(* CODESYS project fablewhole.project
   CompiledLibraryCompatibilityVersion: LeadSysStudio V3.5 SP15 Patch 4
   Title: fablewhole

Project tree, tasks and I/O mapping:
  Device : MC508, Leadshine Technology Co., Ltd., order no. 508101, version 3.5.15.40
      settings: RetainMode = 0; RetainStartAddr = 20480; RetainEndAddr = 524287; RetainSize = 524288; LMMVersion = 0
    application Application
      libraries: Standard, * (System); Util, * (System)
      task T_Motion (cyclic, interval t#4ms, priority 1) calls PRG_Motion
      task T_App (cyclic, interval 20 ms, priority 8) calls PRG_IoMap, PRG_Supervisor, PRG_JobExec, PRG_Test, PRG_Carousels, PRG_Heating, PRG_Sim, PRG_Alarms
      task EtherCAT_Master_Leadshine_A (cyclic, interval 4000 µs, priority 0) calls EtherCAT_Master_Leadshine_A.EtherCAT_Task
      task T_Comms (cyclic, interval 100 ms, priority 15) calls PRG_GatewayComms, PRG_HMI, PRG_HACCP
      01_DUTs/
        data type E_MachMode
        data type E_Item
        data type E_GriddleState
        data type E_FaultClass
        data type ST_Recipe
        data type ST_PattyJob
        data type ST_GriddleSts
        data type ST_TrayInfo
        data type ST_GwCmd
        data type ST_GwAck
        data type ST_AxisSts
        data type ST_HeatZone
        data type ST_Alarm
        data type ST_HaccpRec
        data type ST_MechCmd
      00_GVLs/
        global variables GVL_Cfg
        global variables GVL_Par
        global variables GVL_IO
        global variables GVL_Axes
        global variables GVL_Cmd
        global variables GVL_Sts
        global variables GVL_Alm
        global variables GVL_Mech
      02_L1_Drivers/
        function F_Err [ST]
        function F_RaiseAlarm [ST]
        function block FB_AxisCtrl [ST]
        function block FB_PidHeater [ST]
        function block FB_PneuActuator [ST]
        function block FB_PressDrive [ST]
        function block FB_SensorIn [ST]
        function block FB_VfdIndex [ST]
      03_L2_Mechanisms/
        function block FB_Airlock [ST]
        function block FB_Fork [ST]
        function block FB_FridgeCarousel [ST]
        function block FB_Gantry [ST]
        function block FB_GriddleCarousel [ST]
        function block FB_Gripper [ST]
        function block FB_HeatBank [ST]
        function block FB_IKTransform [ST]
        function block FB_Press [ST]
        function block FB_Refrigeration [ST]
        function block FB_Scraper [ST]
      05_L4_Comms/
        program PRG_Alarms [ST]
        program PRG_GatewayComms [ST]
        program PRG_HACCP [ST]
        program PRG_HMI [ST]
      04_L3_Coordination/
        function block FB_GriddleTracker [ST]
        function block FB_HomingManager [ST]
        function block FB_JobQueue [ST]
        program PRG_JobExec [ST]
        program PRG_Supervisor [ST]
      06_Wiring_Sim_Test/
        program PRG_Carousels [ST]
        program PRG_Heating [ST]
        program PRG_IoMap [ST]
        program PRG_Motion [ST]
        program PRG_Sim [ST]
        program PRG_Test [ST]
    Device Diagnose
    Network Configuration
      LocalBus Config
    Resource Usage
    SoftMotion General Axis Pool
    High_Speed_IO_Module : High Speed IO, Leadshine Technology Co., Ltd., version 3.5.15.40
        unmapped channels: Genral_IO_IN, Genral_IO_Out
    LocalBus_Master_Module : LocalBus Master, Leadshine Technology Co., Ltd., version 3.5.15.40
    EtherCAT_Master_Leadshine_A : EtherCAT Master SoftMotion, 3S - Smart Software Solutions GmbH, version 3.5.15.30
        settings: NetworkName = 'ecat'; SelectNetworkByName = TRUE
      CS3E_D1008 : CS3E-D1008(COE), Leadshine Technology Co.,Ltd., order no. CS3E-D1008, version Revision=16#00000001
          settings: DC sync0 cycletime = 4000; DC sync1 cycletime = 4000
          unmapped channels: Control Word, Profile Target Position, Touch Probe Function, Last Error Code, Status Word, Modes of Operation display, Position Actual Value, Touch Probe Status, Touch Probe 1 Positive Value, Digital Inputs
        Axis : Axis, 3S - Smart Software Solutions GmbH, order no. 0, version 4.6.1.0
            settings: wDriveID = 0; Commisioning.smci.Distance = 100; Commisioning.smci.Velocity = 100; AdrOffset_8010 = 4; BitOffset_8010 = 0; BitLength_8010 = 16; Address_8010 = '%QW2'; Type_8010 = 'UINT'; AddressPointer_8010 = ADR(%QW2); AdrOffset_8020 = 8; BitOffset_8020 = 0; BitLength_8020 = 32; Address_8020 = '%QD2'; Type_8020 = 'DINT'; AddressPointer_8020 = ADR(%QD2); AdrOffset_8030 = 4294967295; BitOffset_8030 = 0; BitLength_8030 = 0; Address_8030 = ''; Type_8030 = ''; AddressPointer_8030 = 0; AdrOffset_8040 = 4294967295; BitOffset_8040 = 0; BitLength_8040 = 0; Address_8040 = ''; Type_8040 = ''; AddressPointer_8040 = 0; AdrOffset_8050 = 4294967295; BitOffset_8050 = 0; BitLength_8050 = 0; Address_8050 = ''; Type_8050 = ''; AddressPointer_8050 = 0; AdrOffset_8060 = 12; BitOffset_8060 = 0; BitLength_8060 = 16; Address_8060 = '%QW6'; Type_8060 = 'UINT'; AddressPointer_8060 = ADR(%QW6); AdrOffset_8070 = 4294967295;
              BitOffset_8070 = 0; BitLength_8070 = 0; Address_8070 = ''; Type_8070 = ''; AddressPointer_8070 = 0; AdrOffset_8080 = 4294967295; BitOffset_8080 = 0; BitLength_8080 = 0; Address_8080 = ''; Type_8080 = ''; AddressPointer_8080 = 0; AdrOffset_8090 = 4294967295; BitOffset_8090 = 0; BitLength_8090 = 0; Address_8090 = ''; Type_8090 = ''; AddressPointer_8090 = 0; AdrOffset_8510 = 6; BitOffset_8510 = 0; BitLength_8510 = 16; Address_8510 = '%IW3'; Type_8510 = 'UINT'; AddressPointer_8510 = ADR(%IW3); AdrOffset_8520 = 12; BitOffset_8520 = 0; BitLength_8520 = 32; Address_8520 = '%ID3'; Type_8520 = 'DINT'; AddressPointer_8520 = ADR(%ID3); AdrOffset_8530 = 4294967295; BitOffset_8530 = 0; BitLength_8530 = 0; Address_8530 = ''; Type_8530 = ''; AddressPointer_8530 = 0; AdrOffset_8540 = 4294967295; BitOffset_8540 = 0; BitLength_8540 = 0; Address_8540 = ''; Type_8540 = '';
              AddressPointer_8540 = 0; AdrOffset_8550 = 8; BitOffset_8550 = 0; BitLength_8550 = 8; Address_8550 = '%IB8'; Type_8550 = 'SINT'; AddressPointer_8550 = ADR(%IB8); AdrOffset_8560 = 24; BitOffset_8560 = 0; BitLength_8560 = 32; Address_8560 = '%ID6'; Type_8560 = 'UDINT'; AddressPointer_8560 = ADR(%ID6); AdrOffset_8570 = 16; BitOffset_8570 = 0; BitLength_8570 = 16; Address_8570 = '%IW8'; Type_8570 = 'UINT'; AddressPointer_8570 = ADR(%IW8); AdrOffset_8580 = 20; BitOffset_8580 = 0; BitLength_8580 = 32; Address_8580 = '%ID5'; Type_8580 = 'DINT'; AddressPointer_8580 = ADR(%ID5); AdrOffset_8590 = 4294967295; BitOffset_8590 = 0; BitLength_8590 = 0; Address_8590 = ''; Type_8590 = ''; AddressPointer_8590 = 0; AdrOffset_8600 = 4294967295; BitOffset_8600 = 0; BitLength_8600 = 0; Address_8600 = ''; Type_8600 = ''; AddressPointer_8600 = 0; AdrOffset_8600 = 4294967295; BitOffset_8600 = 0; BitLength_8600 = 0;
              Address_8610 = ''; Type_8610 = ''; AddressPointer_8610 = 0; AdrOffset_8620 = 4294967295; BitOffset_8620 = 0; BitLength_8620 = 0; Address_8620 = ''; Type_8620 = ''; AddressPointer_8620 = 0
      CS3E_D1008_1 : CS3E-D1008(COE), Leadshine Technology Co.,Ltd., order no. CS3E-D1008, version Revision=16#00000001
          settings: DC sync0 cycletime = 4000; DC sync1 cycletime = 4000
          unmapped channels: Control Word, Profile Target Position, Touch Probe Function, Last Error Code, Status Word, Modes of Operation display, Position Actual Value, Touch Probe Status, Touch Probe 1 Positive Value, Digital Inputs
        Axis_1 : Axis, 3S - Smart Software Solutions GmbH, order no. 0, version 4.6.1.0
            settings: AdrOffset_8010 = 16; BitOffset_8010 = 0; BitLength_8010 = 16; Address_8010 = '%QW8'; Type_8010 = 'UINT'; AddressPointer_8010 = ADR(%QW8); AdrOffset_8020 = 20; BitOffset_8020 = 0; BitLength_8020 = 32; Address_8020 = '%QD5'; Type_8020 = 'DINT'; AddressPointer_8020 = ADR(%QD5); AdrOffset_8030 = 4294967295; BitOffset_8030 = 0; BitLength_8030 = 0; Address_8030 = ''; Type_8030 = ''; AddressPointer_8030 = 0; AdrOffset_8040 = 4294967295; BitOffset_8040 = 0; BitLength_8040 = 0; Address_8040 = ''; Type_8040 = ''; AddressPointer_8040 = 0; AdrOffset_8050 = 4294967295; BitOffset_8050 = 0; BitLength_8050 = 0; Address_8050 = ''; Type_8050 = ''; AddressPointer_8050 = 0; AdrOffset_8060 = 24; BitOffset_8060 = 0; BitLength_8060 = 16; Address_8060 = '%QW12'; Type_8060 = 'UINT'; AddressPointer_8060 = ADR(%QW12); AdrOffset_8070 = 4294967295; BitOffset_8070 = 0; BitLength_8070 = 0; Address_8070 = '';
              Type_8070 = ''; AddressPointer_8070 = 0; AdrOffset_8080 = 4294967295; BitOffset_8080 = 0; BitLength_8080 = 0; Address_8080 = ''; Type_8080 = ''; AddressPointer_8080 = 0; AdrOffset_8090 = 4294967295; BitOffset_8090 = 0; BitLength_8090 = 0; Address_8090 = ''; Type_8090 = ''; AddressPointer_8090 = 0; AdrOffset_8510 = 30; BitOffset_8510 = 0; BitLength_8510 = 16; Address_8510 = '%IW15'; Type_8510 = 'UINT'; AddressPointer_8510 = ADR(%IW15); AdrOffset_8520 = 36; BitOffset_8520 = 0; BitLength_8520 = 32; Address_8520 = '%ID9'; Type_8520 = 'DINT'; AddressPointer_8520 = ADR(%ID9); AdrOffset_8530 = 4294967295; BitOffset_8530 = 0; BitLength_8530 = 0; Address_8530 = ''; Type_8530 = ''; AddressPointer_8530 = 0; AdrOffset_8540 = 4294967295; BitOffset_8540 = 0; BitLength_8540 = 0; Address_8540 = ''; Type_8540 = ''; AddressPointer_8540 = 0; AdrOffset_8550 = 32; BitOffset_8550 = 0;
              BitLength_8550 = 8; Address_8550 = '%IB32'; Type_8550 = 'SINT'; AddressPointer_8550 = ADR(%IB32); AdrOffset_8560 = 48; BitOffset_8560 = 0; BitLength_8560 = 32; Address_8560 = '%ID12'; Type_8560 = 'UDINT'; AddressPointer_8560 = ADR(%ID12); AdrOffset_8570 = 40; BitOffset_8570 = 0; BitLength_8570 = 16; Address_8570 = '%IW20'; Type_8570 = 'UINT'; AddressPointer_8570 = ADR(%IW20); AdrOffset_8580 = 44; BitOffset_8580 = 0; BitLength_8580 = 32; Address_8580 = '%ID11'; Type_8580 = 'DINT'; AddressPointer_8580 = ADR(%ID11); AdrOffset_8590 = 4294967295; BitOffset_8590 = 0; BitLength_8590 = 0; Address_8590 = ''; Type_8590 = ''; AddressPointer_8590 = 0; AdrOffset_8600 = 4294967295; BitOffset_8600 = 0; BitLength_8600 = 0; Address_8600 = ''; Type_8600 = ''; AddressPointer_8600 = 0; AdrOffset_8600 = 4294967295; BitOffset_8600 = 0; BitLength_8600 = 0; Address_8610 = ''; Type_8610 = ''; AddressPointer_8610 = 0;
              AdrOffset_8620 = 4294967295; BitOffset_8620 = 0; BitLength_8620 = 0; Address_8620 = ''; Type_8620 = ''; AddressPointer_8620 = 0
    ModbusCOM_Master_1 : ModbusCOM RS-485 Master, Leadshine Technology Co., Ltd., version 3.5.15.40
        settings: com.Parity = 2; com.Baudrate = 115200
      ModbusCOM_Slave : ModbusCOM Slave, Leadshine Technology Co., Ltd., version 3.5.15.40
          settings: ModBusRTU_ErrorCode = 0; channel 00.FuncCode = 16; channel 00.ControlMode = 1; channel 00.ResendCount = 3; channel 00.WriteRegOffSet = 25089; channel 00.WriteRegLeg = 2; channel 00.IOChannel = 0; channel 00.ChannelName = 'pr0'; channel 00.ChannelNote = ''; channel 01.FuncCode = 16; channel 01.ControlMode = 1; channel 01.ResendCount = 3; channel 01.WriteRegOffSet = 25097; channel 01.WriteRegLeg = 2; channel 01.ChannelName = 'pr1'; channel 01.ChannelNote = ''; channel 02.FuncCode = 16; channel 02.ControlMode = 1; channel 02.ResendCount = 3; channel 02.WriteRegOffSet = 25105; channel 02.WriteRegLeg = 2; channel 02.IOChannel = 2; channel 02.ChannelName = 'pr2'; channel 02.ChannelNote = ''; channel 03.FuncCode = 6; channel 03.ControlMode = 1; channel 03.ResendCount = 1; channel 03.WriteRegOffSet = 24578; channel 03.IOChannel = 3; channel 03.ChannelName = 'hometrig'; channel 03.ChannelNote = ''; channel 04.FuncCode = 3; channel 04.ResendCount = 1; channel 04.ReadRegOffSet = 4099; channel 04.IOChannel = 4; channel 04.ChannelName = 'homestatus'; channel 04.ChannelNote = ''; channel 05.FuncCode = 6; channel 05.ControlMode = 1; channel 05.ResendCount = 1;
            channel 05.WriteRegOffSet = 6145; channel 05.IOChannel = 5; channel 05.ChannelName = 'jog'; channel 05.ChannelNote = ''; Vendor.ChannelNum = 6; Vendor.Timeout = 200
          unmapped channels: ErrorCode, channel 00, channel 00, channel 00, channel 01, channel 01, channel 01, channel 02, channel 02, channel 02, channel 03, channel 03, channel 03, channel 04, channel 04, channel 05, channel 05, channel 05
      ModbusCOM_Slave_1 : ModbusCOM Slave, Leadshine Technology Co., Ltd., version 3.5.15.40
          settings: ModBusRTU_ErrorCode = 0; Vendor.SlaveID = 2
          unmapped channels: ErrorCode
      ModbusCOM_Slave_2 : ModbusCOM Slave, Leadshine Technology Co., Ltd., version 3.5.15.40
          settings: ModBusRTU_ErrorCode = 0; Vendor.SlaveID = 3
          unmapped channels: ErrorCode
      ModbusCOM_Slave_3 : ModbusCOM Slave, Leadshine Technology Co., Ltd., version 3.5.15.40
          settings: ModBusRTU_ErrorCode = 0; Vendor.SlaveID = 4
          unmapped channels: ErrorCode
    ModbusTCP_Slave_Device : Modbus TCP Slave, Leadshine Technology Co., Ltd., version 00.00.00.10
*)

// Device/Application/01_DUTs/E_MachMode
{attribute 'qualified_only'}
{attribute 'strict'}
TYPE E_MachMode :
(
    BOOT    := 0,
    HOMING  := 1,
    READY   := 2,
    RUN     := 3,
    CLEAN   := 4,
    FAULT   := 5,
    ESTOP   := 6
);
END_TYPE

// Device/Application/01_DUTs/E_Item
{attribute 'qualified_only'}
{attribute 'strict'}
TYPE E_Item :
(
    NONE      := 0,
    BEEF      := 1,
    CHICKEN   := 2,
    BACON     := 3,
    PINEAPPLE := 4
);
END_TYPE

// Device/Application/01_DUTs/E_GriddleState
{attribute 'qualified_only'}
{attribute 'strict'}
TYPE E_GriddleState :
(
    EMPTY           := 0,
    LOADING         := 1,
    COOKING         := 2,
    READY_TO_SCRAPE := 3,
    SCRAPING        := 4,
    FAULTED         := 5
);
END_TYPE

// Device/Application/01_DUTs/E_FaultClass
{attribute 'qualified_only'}
{attribute 'strict'}
TYPE E_FaultClass :
(
    INFO         := 0,
    QUARANTINE   := 1,
    ZONE_STOP    := 2,
    MACHINE_STOP := 3
);
END_TYPE

// Device/Application/01_DUTs/ST_Recipe
TYPE ST_Recipe :
STRUCT
    item        : UINT;           // E_Item value
    cookTimeS   : LREAL := 90.0;
    smashDurS   : LREAL := 8.0;
    smashPosMm  : LREAL := 4.0;   // platen gap at smash
    holdPosMm   : LREAL := 6.0;   // light-contact gap for remainder of cook
    platenSetC  : LREAL := 200.0;
END_STRUCT
END_TYPE

// Device/Application/01_DUTs/ST_PattyJob
TYPE ST_PattyJob :
STRUCT
    jobId     : UDINT;
    orderId   : UDINT;
    item      : UINT;
    trayId    : UINT;
    griddleId : INT;
    slot      : INT;
END_STRUCT
END_TYPE

// Device/Application/01_DUTs/ST_GriddleSts
TYPE ST_GriddleSts :
STRUCT
    state        : UINT;   // E_GriddleState value
    item         : UINT;
    count        : INT;
    cookElapsedS : LREAL;
    batchId      : UDINT;
END_STRUCT
END_TYPE

// Device/Application/01_DUTs/ST_TrayInfo
TYPE ST_TrayInfo :
STRUCT
    trayId    : UINT;
    item      : UINT;
    remaining : INT;
    level     : INT;   // 0..19
    face      : INT;   // 0..1
    inChamber : BOOL;
END_STRUCT
END_TYPE

// Device/Application/01_DUTs/ST_GwCmd
TYPE ST_GwCmd :
STRUCT
    seq  : UINT;
    code : UINT;    // see GVL_Cfg CMD_* constants
    p1   : DINT;
    p2   : DINT;
    p3   : DINT;
    p4   : DINT;
END_STRUCT
END_TYPE

// Device/Application/01_DUTs/ST_GwAck
TYPE ST_GwAck :
STRUCT
    seqEcho : UINT;
    busy    : BOOL;
    done    : BOOL;
    error   : BOOL;
    errorId : UDINT;
END_STRUCT
END_TYPE

// Device/Application/01_DUTs/ST_AxisSts
TYPE ST_AxisSts :
STRUCT
    powered : BOOL;
    homed   : BOOL;
    inPos   : BOOL;
    actPos  : LREAL;
    errorId : UDINT;
END_STRUCT
END_TYPE

// Device/Application/01_DUTs/ST_HeatZone
TYPE ST_HeatZone :
STRUCT
    setC    : LREAL;
    actC    : LREAL;
    outPct  : LREAL;
    tcOk    : BOOL;
    atSet   : BOOL;
    enabled : BOOL;
END_STRUCT
END_TYPE

// Device/Application/01_DUTs/ST_Alarm
TYPE ST_Alarm :
STRUCT
    id     : UDINT;      // (subsystem<<16) OR code
    class  : UINT;       // E_FaultClass value
    tsS    : UDINT;      // uptime seconds at raise
    active : BOOL;
    acked  : BOOL;
END_STRUCT
END_TYPE

// Device/Application/01_DUTs/ST_HaccpRec
TYPE ST_HaccpRec :
STRUCT
    batchId    : UDINT;
    item       : UINT;
    griddleId  : INT;
    platenTopC : LREAL;
    platenBotC : LREAL;
    cookS      : LREAL;
    tStartS    : UDINT;
    tEndS      : UDINT;
    result     : UINT;   // 0=OK 1=QUARANTINE
END_STRUCT
END_TYPE

// Device/Application/01_DUTs/ST_MechCmd
TYPE ST_MechCmd :
STRUCT
    code : UINT;    // mechanism-local, see GVL_Cfg MCMD_* constants
    p1   : LREAL;
    p2   : LREAL;
    p3   : LREAL;
END_STRUCT
END_TYPE

// Device/Application/00_GVLs/GVL_Cfg
(* ============================================================
   GVL_Cfg — machine constants. VAR_GLOBAL CONSTANT.
   SIM_MODE is the ONLY switch between simulation and hardware.
   Set FALSE for production download. Never change at runtime.
   ============================================================ *)
VAR_GLOBAL CONSTANT
    SIM_MODE          : BOOL  := TRUE;    // <<< FALSE for real hardware
    SIM_TIME_SCALE    : LREAL := 5.0;     // thermal/cook acceleration in sim (1.0 = real time)

    T_MOTION_MS       : LREAL := 4.0;
    T_APP_MS          : LREAL := 20.0;

    // ---- Counts & geometry ----
    GRIDDLE_COUNT       : INT := 4;
    PATTIES_PER_GRIDDLE : INT := 6;
    STATIONS            : INT := 4;       // carousel stations
    STATION_LOAD        : INT := 0;       // station index where loading happens
    STATION_SCRAPE      : INT := 2;       // opposite station
    TRAY_COLS           : INT := 6;
    TRAY_ROWS           : INT := 4;
    PATTIES_PER_TRAY    : INT := 24;
    TRAY_LEVELS         : INT := 20;
    TRAY_FACES          : INT := 2;

    // ---- Gantry kinematics (mm / deg) ----
    ARM_LEN     : LREAL := 350.0;
    GX_MIN      : LREAL := 0.0;
    GX_MAX      : LREAL := 900.0;
    THETA_MIN   : LREAL := -90.0;
    THETA_MAX   : LREAL := 90.0;
    GZ_UP       : LREAL := 0.0;
    GZ_PICK     : LREAL := 80.0;
    GZ_PLACE    : LREAL := 60.0;
    THETA_SAFE  : LREAL := 0.0;
    GX_PARK     : LREAL := 50.0;
    // tray pick grid (chamber tray held by fork)
    PICK_BASE_X    : LREAL := 700.0;
    PICK_BASE_Y    : LREAL := -150.0;
    PICK_SPACING_X : LREAL := 60.0;
    PICK_SPACING_Y : LREAL := 60.0;
    // griddle place grid (station 0, bottom platen)
    PLACE_BASE_X   : LREAL := 450.0;
    PLACE_BASE_Y   : LREAL := 0.0;
    PLACE_SPC_X    : LREAL := 70.0;
    PLACE_SPC_Y    : LREAL := 70.0;
    PLACE_COLS     : INT   := 3;      // 3 x 2 slots on a griddle

    // ---- Speeds ----
    G_VEL      : LREAL := 400.0;   G_ACC : LREAL := 1500.0;   // gantry X mm/s
    T_VEL      : LREAL := 120.0;   T_ACC : LREAL := 500.0;    // theta deg/s
    Z_VEL      : LREAL := 200.0;   Z_ACC : LREAL := 1000.0;
    S_VEL      : LREAL := 300.0;   S_ACC : LREAL := 1200.0;   // scraper
    F_VEL      : LREAL := 150.0;   F_ACC : LREAL := 400.0;    // fork
    JOG_VEL_MAX: LREAL := 50.0;

    // ---- Recipe edit bounds (PRG_HMI rejects writes outside these) ----
    REC_COOK_MIN   : LREAL := 10.0;   REC_COOK_MAX   : LREAL := 300.0;  // s
    REC_SMDUR_MIN  : LREAL := 0.0;    REC_SMDUR_MAX  : LREAL := 30.0;   // s
    REC_SMPOS_MIN  : LREAL := 2.0;    REC_SMPOS_MAX  : LREAL := 12.0;   // mm gap
    REC_HLPOS_MIN  : LREAL := 3.0;    REC_HLPOS_MAX  : LREAL := 15.0;   // mm gap
    REC_PLSET_MIN  : LREAL := 120.0;  REC_PLSET_MAX  : LREAL := 230.0;  // degC

    // ---- Press PR path parameters ----
    PRESS_OPEN_MM     : LREAL := 60.0;  // path 0 open position (clamshell gap)
    PRESS_TRIM_MAX_MM : LREAL := 2.0;   // per-press calibration trim clamp (+/-)

    // ---- CS2RS press Modbus RTU parameterization (RS485, NetworkConfig channels) ----
    PRESS_BENCH_DRIVE : INT := 0;      // bench: -1 = none; 0..3 = that press drive runs
                                        // REAL (DI motion + Modbus params) while machine is sim
    PRESS_PULSES_PER_MM : LREAL := 1000.0;  // TODO calibrate: drive gear -> pulses per mm gap
    // Channel setup reference (VERIFIED against CS2RS manual 5.4.1) — the
    // registers live in the NetworkConfig channel config, not in code:
    //   write-multiple (FC16), length 2, per path: 0x6201 (path0 pos H/L),
    //   0x6209 (path1), 0x6211 (path2). Trigger reg 0x6002 (unused; DI does motion).

    // ---- Scraper geometry ----
    SC_ENGAGE_Z   : LREAL := 45.0;
    SC_UP_Z       : LREAL := 0.0;
    SC_SWEEP_X0   : LREAL := 100.0;
    SC_SWEEP_X1   : LREAL := 420.0;
    SC_ROW_Y      : ARRAY[0..2] OF LREAL := [0.0, 70.0, 140.0];
    SC_STROKES    : INT := 3;

    // ---- Fork geometry ----
    FORK_LEVEL_H   : LREAL := 90.0;   // mm per tray level
    FORK_Z0        : LREAL := 50.0;
    FORK_MICROLIFT : LREAL := 8.0;
    FORK_TELE_OUT  : LREAL := 300.0;
    FORK_TELE_IN   : LREAL := 0.0;

    // ---- Carousels ----
    ENC_CPR          : DINT := 4096;          // counts per carousel rev
    IDX_SPEED_FAST   : INT  := 300;           // VFD speed ref (raw)
    IDX_SPEED_CREEP  : INT  := 40;
    IDX_DECEL_WIN    : DINT := 300;           // counts before target -> creep
    IDX_STOP_WIN     : DINT := 25;            // counts tolerance to drop pin
    IDX_VERIFY_WIN   : DINT := 40;            // encoder-vs-pin plausibility

    // ---- Heating ----
    HEAT_ZONES     : INT   := 8;
    PWM_WINDOW_MS  : LREAL := 2000.0;
    HEAT_KP        : LREAL := 4.0;
    HEAT_KI        : LREAL := 0.05;           // %/ (degC*s)
    HEAT_AT_BAND   : LREAL := 5.0;            // |err| <= band -> atSet
    HEAT_MAX_STAGGER : INT := 2;              // platens ramping at once
    TC_RATE_MAX    : LREAL := 8.0;            // degC/s plausibility
    FRIDGE_SET_C   : LREAL := 4.0;
    FRIDGE_HYST_C  : LREAL := 1.0;
    FRIDGE_EXC_S   : LREAL := 300.0;          // excursion > 5 min -> QUARANTINE

    // ---- Timeouts ----
    TO_AXIS_MOVE   : TIME := T#15S;
    TO_AXIS_HOME   : TIME := T#40S;
    TO_PNEU        : TIME := T#3S;
    TO_PRESS       : TIME := T#15S;
    TO_INDEX       : TIME := T#25S;
    TO_MECH        : TIME := T#60S;
    SCRAPE_GUARD_S : LREAL := 8.0;
    GW_TIMEOUT_S   : LREAL := 10.0;

    // ---- Command codes: Gateway -> PLC (ST_GwCmd.code) ----
    CMD_NOP         : UINT := 0;
    CMD_FETCH_TRAY  : UINT := 1;   // p1=item p2=level p3=face
    CMD_LOAD_GRIDDLE: UINT := 2;   // p1=griddleId p2=count p3=item
    CMD_SCRAPE      : UINT := 3;   // p1=griddleId
    CMD_RETURN_TRAY : UINT := 4;   // p1=level p2=face
    CMD_CLEAN_MODE  : UINT := 5;
    CMD_ABORT       : UINT := 6;

    // ---- Mechanism-local command codes (ST_MechCmd.code) ----
    MCMD_NONE     : UINT := 0;
    MCMD_HOME     : UINT := 1;
    MCMD_PARK     : UINT := 2;
    MCMD_PICK     : UINT := 10;  // gantry: p1=trayIdx(0..23)
    MCMD_PLACE    : UINT := 11;  // gantry: p1=slot(0..5)
    MCMD_SANITIZE : UINT := 13;
    MCMD_FETCH    : UINT := 20;  // fork: p1=level
    MCMD_RETURN   : UINT := 21;  // fork: p1=level
    MCMD_SWEEP    : UINT := 30;  // scraper: p1=strokeIdx(0..2)
    MCMD_PROFILE  : UINT := 40;  // press: recipe via SetRecipe inputs
    MCMD_OPEN     : UINT := 41;  // press open
    MCMD_GOTO     : UINT := 50;  // carousel: p1=station

    // ---- Subsystem IDs for ErrorID = SHL(ss,16) OR code ----
    SS_GANTRY_X  : UINT := 1;   SS_GANTRY_T : UINT := 2;   SS_GANTRY_Z : UINT := 3;
    SS_SCRAPER_X : UINT := 4;   SS_SCRAPER_Y: UINT := 5;   SS_SCRAPER_Z: UINT := 6;
    SS_FORK_Z    : UINT := 7;   SS_FORK_TELE: UINT := 8;
    SS_PRESS_0   : UINT := 10;  // press n -> 10+n
    SS_GRID_CAR  : UINT := 20;  SS_FRIDGE_CAR : UINT := 21;
    SS_HEAT_0    : UINT := 30;  // zone z -> 30+z
    SS_AIRLOCK   : UINT := 40;  SS_REFRIG   : UINT := 41;
    SS_GANTRY    : UINT := 45;  SS_SCRAPER  : UINT := 46;  SS_FORK : UINT := 47;
    SS_GRIPPER   : UINT := 48;
    SS_JOBEXEC   : UINT := 50;  SS_HOMING   : UINT := 51;
    SS_GWCOMMS   : UINT := 60;  SS_PNEU     : UINT := 61;  SS_SENSOR : UINT := 62;

    // ---- Generic error codes ----
    ERR_NONE      : UINT := 0;
    ERR_TIMEOUT   : UINT := 1;
    ERR_DRIVE     : UINT := 2;
    ERR_NOT_HOMED : UINT := 3;
    ERR_UNREACH   : UINT := 4;   // IK unreachable
    ERR_BAD_CMD   : UINT := 5;
    ERR_INTERLOCK : UINT := 6;
    ERR_PIN       : UINT := 7;   // pin/encoder mismatch
    ERR_SENSOR    : UINT := 8;
    ERR_TC        : UINT := 9;
    ERR_ABORTED   : UINT := 10;
    ERR_BUSY      : UINT := 11;
END_VAR

// Device/Application/00_GVLs/GVL_Par
(* ============================================================
   GVL_Par — retained tunables (recipes, offsets). HMI-writable
   through bounds-checked paths only (PRG_HMI / PRG_GatewayComms).
   ============================================================ *)
VAR_GLOBAL RETAIN
    // Index by E_Item value 0..4; [0] unused
    aRecipe : ARRAY[0..4] OF ST_Recipe :=
        [(item:=0),
         (item:=1, cookTimeS:=90.0,  smashDurS:=8.0, smashPosMm:=4.0, holdPosMm:=6.0, platenSetC:=200.0),  // BEEF
         (item:=2, cookTimeS:=110.0, smashDurS:=8.0, smashPosMm:=5.0, holdPosMm:=7.0, platenSetC:=200.0),  // CHICKEN (validate 74C core!)
         (item:=3, cookTimeS:=60.0,  smashDurS:=0.0, smashPosMm:=8.0, holdPosMm:=8.0, platenSetC:=190.0),  // BACON heat only
         (item:=4, cookTimeS:=45.0,  smashDurS:=0.0, smashPosMm:=8.0, holdPosMm:=8.0, platenSetC:=180.0)]; // PINEAPPLE
    jogVel        : LREAL := 20.0;
    pickOffsetX   : LREAL := 0.0;   // commissioning trims
    pickOffsetY   : LREAL := 0.0;
    placeOffsetX  : LREAL := 0.0;
    placeOffsetY  : LREAL := 0.0;
    // per-press smash/hold position trim, mm (+ = larger gap); HMI-adjustable,
    // clamped to +/- GVL_Cfg.PRESS_TRIM_MAX_MM in PRG_HMI
    pressTrimMm   : ARRAY[0..3] OF LREAL := [0.0, 0.0, 0.0, 0.0];
END_VAR

// Device/Application/00_GVLs/GVL_IO
(* ============================================================
   GVL_IO — the ONLY POU with physical addresses.
   SIM NOTE: in SIM_MODE these are never read/written (PRG_IoMap
   short-circuits). Addresses below are PLACEHOLDERS — replace
   with the real electrical map during panel design (see
   MIGRATION_GUIDE.md step 2) and keep wire numbers in comments.
   ============================================================ *)
VAR_GLOBAL
    // ---- Press drives 1..4 (CS2RS PR mode, DI wiring) ----
    qPressSel0    : ARRAY[0..3] OF BOOL;  // TODO real per-drive addresses
    qPressSel1    : ARRAY[0..3] OF BOOL;
    qPressCtrg    : ARRAY[0..3] OF BOOL;
    qPressEnable  : ARRAY[0..3] OF BOOL;
    iPressInPos   : ARRAY[0..3] OF BOOL;
    iPressAlarm   : ARRAY[0..3] OF BOOL;

    // ---- Pneumatics ----
    qDoorFridgeFront AT %QX4.0 : BOOL;
    qDoorFridgeSide  AT %QX4.1 : BOOL;
    qDoorChamber     AT %QX4.2 : BOOL;
    qPinGriddle      AT %QX4.3 : BOOL;
    qPinFridge       AT %QX4.4 : BOOL;
    qGripper         AT %QX4.5 : BOOL;
    iDoorFrFront_Op  AT %IX3.0 : BOOL;  iDoorFrFront_Cl AT %IX3.1 : BOOL;
    iDoorFrSide_Op   AT %IX3.2 : BOOL;  iDoorFrSide_Cl  AT %IX3.3 : BOOL;
    iDoorChamber_Op  AT %IX3.4 : BOOL;  iDoorChamber_Cl AT %IX3.5 : BOOL;
    iPinGriddle_Ext  AT %IX3.6 : BOOL;  iPinGriddle_Ret AT %IX3.7 : BOOL;
    iPinFridge_Ext   AT %IX4.0 : BOOL;  iPinFridge_Ret  AT %IX4.1 : BOOL;
    iGripAcquired    AT %IX4.2 : BOOL;

    // ---- Carousel VFDs (hardwired run/dir + analog/comms speed) ----
    qGridCarFwd AT %QX5.0 : BOOL;  qGridCarRev AT %QX5.1 : BOOL;
    qFrCarFwd   AT %QX5.2 : BOOL;  qFrCarRev   AT %QX5.3 : BOOL;
    wGridCarSpeed AT %QW10 : INT;  wFrCarSpeed  AT %QW11 : INT;
    diGridCarEnc  AT %ID12 : DINT; diFrCarEnc   AT %ID14 : DINT;
    iGridCarHome  AT %IX5.0 : BOOL; iFrCarHome  AT %IX5.1 : BOOL;

    // ---- Heating (R2 modules) ----
    qSsr         : ARRAY[0..7] OF BOOL;
    wPlatenTemp AT %IW20  : ARRAY[0..7] OF INT;   // 0.1 degC
    wFridgeTemp AT %IW28  : INT;                  // 0.1 degC

    // ---- BENCH press-drive terminals (old-rig wiring; PRESS_BENCH_DRIVE=0) ----
    qBenchPrAdd0    AT %QX1.5 : BOOL;  // drive SI = ADD0 (ex Z_DO_Down)
    qBenchPrAdd1    AT %QX1.7 : BOOL;  // drive SI = ADD1 (rewired)
    qBenchPrCtrg    AT %QX1.6 : BOOL;  // drive SI = CTRG (ex Z_Trig)
    qBenchPrDisable AT %QX1.3 : BOOL;  // drive enable line, INVERTED: TRUE = disable (ex Z_Disable)
    iBenchPrInPos   AT %IX1.0 : BOOL;  // SO1 INP (ex Z_InPos)
    iBenchPrAlarm   AT %IX1.1 : BOOL;  // SO3 ALM (ex Z_Alarm — check polarity!)

    // ---- RS485 Modbus master channel image (press PR position writes) ----
    // PLACEHOLDER addresses: after creating the 3 write channels in
    // NetworkConfig (RS485 -> Modbus Master), set these to the addresses the
    // master's I/O mapping actually assigns (old-project pattern: data words
    // %QW, trigger bit %QX, done bit %IX, error word %IW).
    qMbPr0Data AT %QW13 : ARRAY[0..1] OF WORD;  // CH0: slave1 FC16 25089/0x6201 len2 (path0 pos H,L)
    qMbPr1Data AT %QW16 : ARRAY[0..1] OF WORD;  // CH1: slave1 FC16 25097/0x6209 len2 (path1)
    qMbPr2Data AT %QW19 : ARRAY[0..1] OF WORD;  // CH2: slave1 FC16 25105/0x6211 len2 (path2)
    qMbPr0Trig AT %QX30.0 : BOOL;               // trigger control bits
    qMbPr1Trig AT %QX36.0 : BOOL;
    qMbPr2Trig AT %QX42.0 : BOOL;
    iMbPr0Done AT %IX54.0 : BOOL;               // processing complete states
    iMbPr1Done AT %IX54.1 : BOOL;
    iMbPr2Done AT %IX54.2 : BOOL;
    iMbPrErr   AT %IW26   : WORD;               // master ErrorCode (0 = ok)
    // homing + status channels
    qMbPrHomeData AT %QW22   : WORD;            // CH3: slave1 FC06 0x6002/24578 len1 (0x0020 = home)
    qMbPrHomeTrig AT %QX46.0 : BOOL;
    iMbPrHomeDone AT %IX54.3 : BOOL;
    iMbPrStatus   AT %IW28   : WORD;            // CH4: slave1 FC03 0x1003/4099 len1, CYCLE 100ms
    // jog channel (mapped)
    qMbPrJogData AT %QW24   : WORD;             // CH5: slave1 FC06 0x1801/6145 len1 (0x4001/0x4002)
    qMbPrJogTrig AT %QX50.0 : BOOL;
    iMbPrJogDone AT %IX58.1 : BOOL;
                                                // bits: 0x01 fault 0x02 enabled 0x04 running
                                                //       0x20 path done 0x40 homing done

    // ---- Fork brake ----
    qForkBrakeRelease AT %QX7.0 : BOOL;
    iForkBrakeOk      AT %IX6.0 : BOOL;
    iForkTrayPresent  AT %IX6.1 : BOOL;

    // ---- Safety controller status (monitor only) ----
    iSafetyOk        AT %IX7.0 : BOOL;
    iZonePwrMotion   AT %IX7.1 : BOOL;
    iZonePwrPress    AT %IX7.2 : BOOL;
END_VAR

// Device/Application/00_GVLs/GVL_Axes
(* ============================================================
   GVL_Axes — SoftMotion axis references.
   SIMULATION BUILD: the dummy declarations below let the project
   compile with SM3_Basic present but no drives; FB_AxisCtrl never
   calls MC_* while SIM_MODE=TRUE.
   PRODUCTION BUILD: DELETE these dummies and pass the device-tree
   axis objects (names created by the EtherCAT config) directly in
   PRG_Motion — see MIGRATION_GUIDE.md step 3.
   ============================================================ *)
VAR_GLOBAL
    axRefGantryX  : AXIS_REF_SM3;
    axRefGantryT  : AXIS_REF_SM3;
    axRefGantryZ  : AXIS_REF_SM3;
    axRefScraperX : AXIS_REF_SM3;
    axRefScraperY : AXIS_REF_SM3;
    axRefScraperZ : AXIS_REF_SM3;
    axRefForkZ    : AXIS_REF_SM3;
    axRefForkTele : AXIS_REF_SM3;
END_VAR

// Device/Application/00_GVLs/GVL_Cmd
(* ============================================================
   GVL_Cmd — commands INTO the PLC (Gateway + HMI + test).
   Modbus-TCP register images live here (%MW). The MC508 Modbus
   TCP slave exposes %MW to the Gateway.
   ============================================================ *)
VAR_GLOBAL
    // Gateway command image (Modbus 40001..) — packed by PRG_GatewayComms
    mbCmdRegs AT %MW0  : ARRAY[0..9]  OF WORD;   // seq,code,p1..p4 (DINT lo/hi)
    mbAckRegs AT %MW10 : ARRAY[0..5]  OF WORD;
    mbStsRegs AT %MW20 : ARRAY[0..79] OF WORD;
    mbParRegs AT %MW500: ARRAY[0..59] OF WORD;

    gwCmd     : ST_GwCmd;        // decoded, latched command
    gwAck     : ST_GwAck;
    gwHeartbeatIn : UINT;        // written by Gateway (reg in mbCmdRegs[9])
    gwAlive   : BOOL;
    gwPending : BOOL;            // new latched command awaiting JobExec

    // HMI request bits (edge-processed in PRG_HMI)
    hmiStart, hmiStop, hmiReset, hmiAck, hmiClean : BOOL;
    hmiMaintPin : UINT;          // maintenance password value
    hmiJogAxis  : INT;           // 0=none 1..8
    hmiJogPlus, hmiJogMinus : BOOL;

    // HMI recipe editor (bounds-checked in PRG_HMI; rejected in RUN)
    hmiRecItem  : UINT;          // 1..4 = E_Item to edit
    hmiRecField : UINT;          // 1=cookTimeS 2=smashDurS 3=smashPosMm 4=holdPosMm 5=platenSetC
    hmiRecValue : LREAL;         // requested value
    hmiRecWrite : BOOL;          // rising edge applies
    hmiRecAck   : BOOL;          // feedback: accepted
    hmiRecErr   : BOOL;          // feedback: rejected (bounds / mode / index)

    // HMI press calibration trim (maintenance PIN required)
    hmiTrimPress : UINT;         // 0..3
    hmiTrimDelta : LREAL;        // +/- mm added to that press's trim
    hmiTrimWrite : BOOL;         // rising edge applies
    hmiTrimAck, hmiTrimErr : BOOL;

    // HMI press service commands (PIN-gated; bench/commissioning + maintenance)
    hmiPressSel   : UINT;        // 0..3
    hmiPressCmd   : UINT;        // 1=HOME 2=OPEN 3=PROFILE(uses hmiRecItem's recipe)
    hmiPressWrite : BOOL;        // rising edge executes
    hmiPressAck, hmiPressErr : BOOL;

    // LT2100E Modbus-TCP register image (see HMI_LT2100E_GUIDE.md)
    // HMI writes 600..609, reads 620..669. Packed/unpacked in PRG_HMI.
    hmiRegsCmd AT %MW600 : ARRAY[0..9]  OF WORD;
    hmiRegsSts AT %MW620 : ARRAY[0..49] OF WORD;

    // Processed requests to Supervisor
    reqStart, reqStop, reqReset, reqClean, reqAckAll : BOOL;

    // Test authority: PRG_Test drives mechanisms instead of JobExec
    testMode  : BOOL := TRUE;    // default TRUE in sim; set FALSE for gateway runs
    testStart : BOOL;            // rising edge starts the automated suite
END_VAR

// Device/Application/00_GVLs/GVL_Sts
(* ============================================================
   GVL_Sts — status OUT of the PLC + Supervisor coordination
   flags. Written by L2/L3 only; L4 reads.
   ============================================================ *)
VAR_GLOBAL
    mode        : E_MachMode := E_MachMode.BOOT;
    uptimeS     : UDINT;
    heartbeat   : UINT;
    // Supervisor coordination (read by owner PRGs each cycle)
    safetyOk    : BOOL;          // effective (sim: TRUE)
    enMotion    : BOOL;          // mechanisms may move
    enProcess   : BOOL;          // heat + refrigeration on
    abortAll    : BOOL;          // broadcast abort
    resetPulse  : BOOL;          // 1-cycle axis reset on FAULT->HOMING
    cleanCoolOk : BOOL;          // all platens < 60 C in CLEAN
    // Aggregates
    allHomed    : BOOL;
    heatAtSet   : BOOL;
    fridgeAtSet : BOOL;
    fridgeActC  : LREAL;
    aGriddle    : ARRAY[0..3] OF ST_GriddleSts;
    aHeat       : ARRAY[0..7] OF ST_HeatZone;
    tray        : ST_TrayInfo;
    pattyOnGriddle : ARRAY[0..3, 0..5] OF BOOL;  // process bookkeeping (v1: no optics)
    carGridStation : INT;
    carFridgeFace  : INT;
    haccpCount  : UDINT;
    lastHaccp   : ST_HaccpRec;
    activeAlarms: INT;
    gwSilent    : BOOL;
END_VAR

// Device/Application/00_GVLs/GVL_Alm
(* ============================================================
   GVL_Alm — alarm table + history. Managed by PRG_Alarms and
   F_RaiseAlarm (any POU may raise).
   ============================================================ *)
VAR_GLOBAL
    aActive  : ARRAY[0..63] OF ST_Alarm;
    nActive  : INT;
    worstClass : UINT;                 // highest active E_FaultClass
    reqZoneStop : BOOL;                // aggregated flags for Supervisor
    reqMachStop : BOOL;
END_VAR
VAR_GLOBAL RETAIN
    aHistory : ARRAY[0..199] OF ST_Alarm;
    histHead : INT;
END_VAR

// Device/Application/00_GVLs/GVL_Mech
(* ============================================================
   GVL_Mech — ALL FB instances live here (single ownership table).
   BODY-CALL OWNERSHIP (call the FB body ONLY in the listed PRG):
     PRG_Motion   (T_Motion): axis FBs, fbGantry, fbScraper, fbFork, fbGripper
     PRG_Carousels(T_App)   : press drives, presses, VFDs, carousels,
                              pneumatics, airlock
     PRG_Heating  (T_App)   : heaters, heat bank, refrigeration
   All other POUs only WRITE inputs / READ outputs of these instances.
   ============================================================ *)
VAR_GLOBAL
    // L1 axis drivers
    axGX, axGT, axGZ : FB_AxisCtrl;      // gantry X / theta / Z
    axSX, axSY, axSZ : FB_AxisCtrl;      // scraper
    axFZ, axFT       : FB_AxisCtrl;      // fork Z / telescope

    // L1 press drives + L2 presses
    drvPress : ARRAY[0..3] OF FB_PressDrive;
    fbPress  : ARRAY[0..3] OF FB_Press;

    // Pneumatics
    fbDoorFridgeFront, fbDoorFridgeSide, fbDoorChamber : FB_PneuActuator;
    fbPinGriddle, fbPinFridge, fbPneuGrip : FB_PneuActuator;

    // Carousels
    vfdGriddle, vfdFridge : FB_VfdIndex;
    fbGridCar  : FB_GriddleCarousel;
    fbFridgeCar: FB_FridgeCarousel;

    // Heating / cold
    fbHeater  : ARRAY[0..7] OF FB_PidHeater;
    fbHeatBank: FB_HeatBank;
    fbRefrig  : FB_Refrigeration;

    // Motion mechanisms
    fbIK      : FB_IKTransform;
    fbGripper : FB_Gripper;
    fbGantry  : FB_Gantry;
    fbScraper : FB_Scraper;
    fbFork    : FB_Fork;

    // Coordination
    fbAirlock : FB_Airlock;
    fbHoming  : FB_HomingManager;
    fbTracker : FB_GriddleTracker;
    fbQueue   : FB_JobQueue;
END_VAR

// Device/Application/06_Wiring_Sim_Test/PRG_Motion
(* ============================================================
   PRG_Motion — T_Motion (4 ms). Body-call owner for all axis FBs
   and the motion mechanisms. THE ONLY TASK TOUCHING MC_* / AXIS_REF.
   This is the ST equivalent of the CFC wiring diagram: pure
   parameter assignment + instance calls, no logic.
   MIGRATION: replace GVL_Axes.axRef* with the device-tree axis
   objects created by the EtherCAT scan (step 3 of the guide).
   ============================================================ *)
PROGRAM PRG_Motion
VAR
    init : BOOL;
END_VAR

IF NOT init THEN
    init := TRUE;
    GVL_Mech.axGX.SubsysId := GVL_Cfg.SS_GANTRY_X;   GVL_Mech.axGX.CycleMs := GVL_Cfg.T_MOTION_MS;
    GVL_Mech.axGT.SubsysId := GVL_Cfg.SS_GANTRY_T;   GVL_Mech.axGT.CycleMs := GVL_Cfg.T_MOTION_MS;
    GVL_Mech.axGZ.SubsysId := GVL_Cfg.SS_GANTRY_Z;   GVL_Mech.axGZ.CycleMs := GVL_Cfg.T_MOTION_MS;
    GVL_Mech.axSX.SubsysId := GVL_Cfg.SS_SCRAPER_X;  GVL_Mech.axSX.CycleMs := GVL_Cfg.T_MOTION_MS;
    GVL_Mech.axSY.SubsysId := GVL_Cfg.SS_SCRAPER_Y;  GVL_Mech.axSY.CycleMs := GVL_Cfg.T_MOTION_MS;
    GVL_Mech.axSZ.SubsysId := GVL_Cfg.SS_SCRAPER_Z;  GVL_Mech.axSZ.CycleMs := GVL_Cfg.T_MOTION_MS;
    GVL_Mech.axFZ.SubsysId := GVL_Cfg.SS_FORK_Z;     GVL_Mech.axFZ.CycleMs := GVL_Cfg.T_MOTION_MS;
    GVL_Mech.axFT.SubsysId := GVL_Cfg.SS_FORK_TELE;  GVL_Mech.axFT.CycleMs := GVL_Cfg.T_MOTION_MS;
END_IF

// ---- distribute enables / abort / reset ----
GVL_Mech.axGX.Sim := GVL_Cfg.SIM_MODE;  GVL_Mech.axGX.Enable := GVL_Sts.enMotion;
GVL_Mech.axGT.Sim := GVL_Cfg.SIM_MODE;  GVL_Mech.axGT.Enable := GVL_Sts.enMotion;
GVL_Mech.axGZ.Sim := GVL_Cfg.SIM_MODE;  GVL_Mech.axGZ.Enable := GVL_Sts.enMotion;
GVL_Mech.axSX.Sim := GVL_Cfg.SIM_MODE;  GVL_Mech.axSX.Enable := GVL_Sts.enMotion;
GVL_Mech.axSY.Sim := GVL_Cfg.SIM_MODE;  GVL_Mech.axSY.Enable := GVL_Sts.enMotion;
GVL_Mech.axSZ.Sim := GVL_Cfg.SIM_MODE;  GVL_Mech.axSZ.Enable := GVL_Sts.enMotion;
GVL_Mech.axFZ.Sim := GVL_Cfg.SIM_MODE;  GVL_Mech.axFZ.Enable := GVL_Sts.enMotion;
GVL_Mech.axFT.Sim := GVL_Cfg.SIM_MODE;  GVL_Mech.axFT.Enable := GVL_Sts.enMotion;
GVL_Mech.axGX.Abort := GVL_Sts.abortAll;  GVL_Mech.axGX.ResetExec := GVL_Sts.resetPulse;
GVL_Mech.axGT.Abort := GVL_Sts.abortAll;  GVL_Mech.axGT.ResetExec := GVL_Sts.resetPulse;
GVL_Mech.axGZ.Abort := GVL_Sts.abortAll;  GVL_Mech.axGZ.ResetExec := GVL_Sts.resetPulse;
GVL_Mech.axSX.Abort := GVL_Sts.abortAll;  GVL_Mech.axSX.ResetExec := GVL_Sts.resetPulse;
GVL_Mech.axSY.Abort := GVL_Sts.abortAll;  GVL_Mech.axSY.ResetExec := GVL_Sts.resetPulse;
GVL_Mech.axSZ.Abort := GVL_Sts.abortAll;  GVL_Mech.axSZ.ResetExec := GVL_Sts.resetPulse;
GVL_Mech.axFZ.Abort := GVL_Sts.abortAll;  GVL_Mech.axFZ.ResetExec := GVL_Sts.resetPulse;
GVL_Mech.axFT.Abort := GVL_Sts.abortAll;  GVL_Mech.axFT.ResetExec := GVL_Sts.resetPulse;

// ---- mechanism bodies (write axis inputs) ----
GVL_Mech.fbGripper(
    Sim  := GVL_Cfg.SIM_MODE,
    iAcquired := GVL_IO.iGripAcquired,
    Pneu := GVL_Mech.fbPneuGrip);

GVL_Mech.fbGantry(
    Enable := GVL_Sts.enMotion,
    Abort  := GVL_Sts.abortAll,
    Sim    := GVL_Cfg.SIM_MODE,
    AxX := GVL_Mech.axGX, AxT := GVL_Mech.axGT, AxZ := GVL_Mech.axGZ,
    Grip := GVL_Mech.fbGripper, IK := GVL_Mech.fbIK);

GVL_Mech.fbScraper(
    Enable := GVL_Sts.enMotion,
    Abort  := GVL_Sts.abortAll,
    Sim    := GVL_Cfg.SIM_MODE,
    AxX := GVL_Mech.axSX, AxY := GVL_Mech.axSY, AxZ := GVL_Mech.axSZ);

GVL_Mech.fbFork(
    Enable := GVL_Sts.enMotion,
    Abort  := GVL_Sts.abortAll,
    Sim    := GVL_Cfg.SIM_MODE,
    iBrakeOk := GVL_IO.iForkBrakeOk,
    iTrayPresent := GVL_IO.iForkTrayPresent,
    AxZ := GVL_Mech.axFZ, AxT := GVL_Mech.axFT);
IF NOT GVL_Cfg.SIM_MODE THEN
    GVL_IO.qForkBrakeRelease := GVL_Mech.fbFork.qBrakeRelease;
END_IF

// ---- axis bodies LAST (consume inputs written above) ----
GVL_Mech.axGX(Axis := GVL_Axes.axRefGantryX);
GVL_Mech.axGT(Axis := GVL_Axes.axRefGantryT);
GVL_Mech.axGZ(Axis := GVL_Axes.axRefGantryZ);
GVL_Mech.axSX(Axis := GVL_Axes.axRefScraperX);
GVL_Mech.axSY(Axis := GVL_Axes.axRefScraperY);
GVL_Mech.axSZ(Axis := GVL_Axes.axRefScraperZ);
GVL_Mech.axFZ(Axis := GVL_Axes.axRefForkZ);
GVL_Mech.axFT(Axis := GVL_Axes.axRefForkTele);

END_PROGRAM

// Device/Application/06_Wiring_Sim_Test/PRG_IoMap
(* ============================================================
   PRG_IoMap — T_App, runs FIRST. Housekeeping + the place for
   commissioning force-rungs (these networks become LD at the
   language refactor). All %I/%Q symbol reads/writes elsewhere go
   through the owner wiring PRGs; addresses exist ONLY in GVL_IO.
   ============================================================ *)
PROGRAM PRG_IoMap
VAR
    msAcc : LREAL;
END_VAR

msAcc := msAcc + GVL_Cfg.T_APP_MS;
IF msAcc >= 1000.0 THEN
    msAcc := msAcc - 1000.0;
    GVL_Sts.uptimeS := GVL_Sts.uptimeS + 1;
END_IF
// ---- bench press-drive terminal mapping (active when PRESS_BENCH_DRIVE = 0) ----
// Copies the unaddressed press-0 signal arrays to/from the physically wired
// bench terminals (declared in GVL_IO, old-rig addresses).
IF GVL_Cfg.PRESS_BENCH_DRIVE = 0 THEN
    GVL_IO.qBenchPrAdd0    := GVL_IO.qPressSel0[0];
    GVL_IO.qBenchPrAdd1    := GVL_IO.qPressSel1[0];
    GVL_IO.qBenchPrCtrg    := GVL_IO.qPressCtrg[0];
    GVL_IO.qBenchPrDisable := NOT GVL_IO.qPressEnable[0];   // wire is a DISABLE line
    GVL_IO.iPressInPos[0]  := GVL_IO.iBenchPrInPos;
    GVL_IO.iPressAlarm[0]  := GVL_IO.iBenchPrAlarm;         // if ALM is NC: invert here
END_IF

// TODO(commissioning): add per-signal force flags here, e.g.
//   IF forceDoorChamber THEN GVL_IO.qDoorChamber := forceVal; END_IF

END_PROGRAM

// Device/Application/04_L3_Coordination/PRG_Supervisor
(* ============================================================
   PRG_Supervisor — machine mode state machine (T_App, runs FIRST
   among coordinators). Owns: mode transitions, enable distribution,
   abort broadcast, homing orchestration, clean-mode thermal gate.
   Safety is only MONITORED here (GVL_Sts.safetyOk).
   ============================================================ *)
PROGRAM PRG_Supervisor
VAR
    rtStart, rtStop, rtReset, rtClean : R_TRIG;
    z          : INT;
    coolOk     : BOOL;
    firstScan  : BOOL := TRUE;
END_VAR

// effective safety status
GVL_Sts.safetyOk := GVL_Cfg.SIM_MODE OR GVL_IO.iSafetyOk;

rtStart(CLK := GVL_Cmd.reqStart);
rtStop (CLK := GVL_Cmd.reqStop);
rtReset(CLK := GVL_Cmd.reqReset);
rtClean(CLK := GVL_Cmd.reqClean);

// defaults each scan
GVL_Sts.resetPulse := FALSE;

// global overrides
IF NOT GVL_Sts.safetyOk THEN
    GVL_Sts.mode := E_MachMode.ESTOP;
END_IF
IF GVL_Alm.reqMachStop AND (GVL_Sts.mode <> E_MachMode.ESTOP) THEN
    GVL_Sts.mode := E_MachMode.FAULT;
END_IF

CASE GVL_Sts.mode OF
    E_MachMode.BOOT:
        GVL_Sts.enMotion := FALSE; GVL_Sts.enProcess := FALSE;
        GVL_Sts.abortAll := FALSE;
        IF GVL_Sts.safetyOk AND NOT firstScan THEN
            GVL_Sts.resetPulse := TRUE;
            GVL_Mech.fbHoming.Exec := TRUE;
            GVL_Sts.mode := E_MachMode.HOMING;
        END_IF

    E_MachMode.HOMING:
        GVL_Sts.enMotion := TRUE; GVL_Sts.enProcess := FALSE;
        IF GVL_Mech.fbHoming.Done THEN
            GVL_Mech.fbHoming.Exec := FALSE;
            GVL_Sts.mode := E_MachMode.READY;
        ELSIF GVL_Mech.fbHoming.Error THEN
            GVL_Mech.fbHoming.Exec := FALSE;
            GVL_Sts.mode := E_MachMode.FAULT;
        END_IF

    E_MachMode.READY:
        GVL_Sts.enMotion := TRUE; GVL_Sts.enProcess := TRUE;   // heat-up + pulldown
        IF GVL_Alm.reqZoneStop THEN
            GVL_Sts.mode := E_MachMode.FAULT;
        ELSIF rtStart.Q AND GVL_Sts.heatAtSet AND GVL_Sts.fridgeAtSet AND GVL_Sts.allHomed THEN
            GVL_Sts.mode := E_MachMode.RUN;
        END_IF

    E_MachMode.RUN:
        GVL_Sts.enMotion := TRUE; GVL_Sts.enProcess := TRUE;
        IF GVL_Alm.reqZoneStop THEN
            GVL_Sts.mode := E_MachMode.FAULT;
        ELSIF rtStop.Q THEN
            GVL_Sts.mode := E_MachMode.READY;      // finish-in-place is JobExec's job
        ELSIF rtClean.Q AND (GVL_Mech.fbQueue.Empty) THEN
            GVL_Sts.mode := E_MachMode.CLEAN;
        END_IF

    E_MachMode.CLEAN:
        GVL_Sts.enMotion := FALSE;                  // motion locked for operator
        GVL_Sts.enProcess := FALSE;                 // heaters off -> cool down
        coolOk := TRUE;
        FOR z := 0 TO 7 DO
            IF GVL_Sts.aHeat[z].actC >= 60.0 THEN coolOk := FALSE; END_IF
        END_FOR
        GVL_Sts.cleanCoolOk := coolOk;
        IF rtStart.Q AND coolOk THEN                // operator confirms clean done
            GVL_Sts.resetPulse := TRUE;
            GVL_Mech.fbHoming.Exec := TRUE;
            GVL_Sts.mode := E_MachMode.HOMING;
        END_IF

    E_MachMode.FAULT:
        GVL_Sts.enMotion := FALSE; GVL_Sts.enProcess := FALSE;
        GVL_Sts.abortAll := TRUE;
        IF rtReset.Q AND (NOT GVL_Alm.reqMachStop) AND (NOT GVL_Alm.reqZoneStop) THEN
            GVL_Sts.abortAll := FALSE;
            GVL_Sts.resetPulse := TRUE;
            GVL_Mech.fbHoming.Exec := TRUE;
            GVL_Sts.mode := E_MachMode.HOMING;
        END_IF

    E_MachMode.ESTOP:
        GVL_Sts.enMotion := FALSE; GVL_Sts.enProcess := FALSE;
        GVL_Sts.abortAll := TRUE;
        IF GVL_Sts.safetyOk AND rtReset.Q THEN
            GVL_Sts.abortAll := FALSE;
            GVL_Sts.resetPulse := TRUE;
            GVL_Mech.fbHoming.Exec := TRUE;
            GVL_Sts.mode := E_MachMode.HOMING;
        END_IF
END_CASE
firstScan := FALSE;

// homing manager body (same task, before PRG_Carousels)
GVL_Mech.fbHoming(
    Abort     := GVL_Sts.abortAll,
    Presses   := GVL_Mech.fbPress,
    Gantry    := GVL_Mech.fbGantry,
    Scraper   := GVL_Mech.fbScraper,
    Fork      := GVL_Mech.fbFork,
    GridCar   := GVL_Mech.fbGridCar,
    FridgeCar := GVL_Mech.fbFridgeCar);

// aggregates
GVL_Sts.allHomed := GVL_Mech.fbGantry.Homed AND GVL_Mech.fbScraper.Homed
                AND GVL_Mech.fbFork.Homed AND GVL_Mech.fbGridCar.Homed
                AND GVL_Mech.fbFridgeCar.Homed;
GVL_Sts.heatAtSet   := GVL_Mech.fbHeatBank.AllAtSet;
GVL_Sts.fridgeAtSet := GVL_Mech.fbRefrig.AtSet;
GVL_Sts.fridgeActC  := GVL_Mech.fbRefrig.ActC;

END_PROGRAM

// Device/Application/06_Wiring_Sim_Test/PRG_Carousels
(* ============================================================
   PRG_Carousels — T_App body-call owner: press drives, presses,
   pneumatics, VFD indexers, carousels, airlock. Pure wiring
   (the ST equivalent of a CFC sheet). Runs AFTER Supervisor/
   JobExec/Test (which write the Cmd inputs).
   ============================================================ *)
PROGRAM PRG_Carousels
VAR
    i    : INT;
    init : BOOL;
END_VAR

IF NOT init THEN
    init := TRUE;
    FOR i := 0 TO 3 DO
        GVL_Mech.drvPress[i].SubsysId := GVL_Cfg.SS_PRESS_0 + TO_UINT(i);
        GVL_Mech.fbPress[i].PressId := i;
    END_FOR
    GVL_Mech.fbDoorFridgeFront.SubsysId := GVL_Cfg.SS_AIRLOCK;
    GVL_Mech.fbDoorFridgeSide.SubsysId  := GVL_Cfg.SS_AIRLOCK;
    GVL_Mech.fbDoorChamber.SubsysId     := GVL_Cfg.SS_AIRLOCK;
    GVL_Mech.fbPinGriddle.SubsysId := GVL_Cfg.SS_GRID_CAR;
    GVL_Mech.fbPinFridge.SubsysId  := GVL_Cfg.SS_FRIDGE_CAR;
    GVL_Mech.fbPneuGrip.SubsysId   := GVL_Cfg.SS_GRIPPER;
    GVL_Mech.vfdGriddle.SubsysId := GVL_Cfg.SS_GRID_CAR;
    GVL_Mech.vfdFridge.SubsysId  := GVL_Cfg.SS_FRIDGE_CAR;
END_IF

// ---- presses ----
FOR i := 0 TO 3 DO
    GVL_Mech.fbPress[i].Enable := GVL_Sts.enMotion;
    GVL_Mech.fbPress[i].Abort  := GVL_Sts.abortAll;
    GVL_Mech.fbPress[i].Sim    := GVL_Cfg.SIM_MODE;
    GVL_Mech.fbPress[i].CycleMs:= GVL_Cfg.T_APP_MS;
    // bench override: the selected drive runs REAL while the machine is sim
    GVL_Mech.drvPress[i].Sim    := GVL_Cfg.SIM_MODE AND (i <> GVL_Cfg.PRESS_BENCH_DRIVE);
    GVL_Mech.drvPress[i].Enable := GVL_Sts.enMotion;
    GVL_Mech.drvPress[i].Abort  := GVL_Sts.abortAll;
    GVL_Mech.drvPress[i].CycleMs:= GVL_Cfg.T_APP_MS;
    GVL_Mech.drvPress[i].iInPos := GVL_IO.iPressInPos[i];
    GVL_Mech.drvPress[i].iAlarm := GVL_IO.iPressAlarm[i];
    GVL_Mech.fbPress[i](Drv := GVL_Mech.drvPress[i]);
    GVL_Mech.drvPress[i]();
    IF (NOT GVL_Cfg.SIM_MODE) OR (i = GVL_Cfg.PRESS_BENCH_DRIVE) THEN
        GVL_IO.qPressSel0[i]   := GVL_Mech.drvPress[i].qSel0;
        GVL_IO.qPressSel1[i]   := GVL_Mech.drvPress[i].qSel1;
        GVL_IO.qPressCtrg[i]   := GVL_Mech.drvPress[i].qCtrg;
        GVL_IO.qPressEnable[i] := GVL_Mech.drvPress[i].qEnable;
    END_IF
END_FOR

// ---- CS2RS Modbus PR-write transport: NetworkConfig channel routing ----
// Channels are created in NetworkConfig (RS485 -> Modbus Master), one
// write-multiple channel per PR path (see GVL_IO placeholders + GVL_Cfg
// reference). This glue routes the bench/press-0 drive's path-write request
// to the matching channel. Extend with channel banks for drives 1..3 when
// the full RS485 bus exists.
IF (NOT GVL_Cfg.SIM_MODE) OR (GVL_Cfg.PRESS_BENCH_DRIVE >= 0) THEN
    GVL_IO.qMbPr0Trig := FALSE;
    GVL_IO.qMbPr1Trig := FALSE;
    GVL_IO.qMbPr2Trig := FALSE;
    GVL_Mech.drvPress[0].MbWrDone := FALSE;
    GVL_Mech.drvPress[0].MbWrErr  := FALSE;
    CASE GVL_Mech.drvPress[0].MbPath OF
        0:  GVL_IO.qMbPr0Data[0] := GVL_Mech.drvPress[0].MbValH;
            GVL_IO.qMbPr0Data[1] := GVL_Mech.drvPress[0].MbValL;
            GVL_IO.qMbPr0Trig    := GVL_Mech.drvPress[0].MbWrExec;
            GVL_Mech.drvPress[0].MbWrDone := GVL_IO.iMbPr0Done AND GVL_Mech.drvPress[0].MbWrExec;
        1:  GVL_IO.qMbPr1Data[0] := GVL_Mech.drvPress[0].MbValH;
            GVL_IO.qMbPr1Data[1] := GVL_Mech.drvPress[0].MbValL;
            GVL_IO.qMbPr1Trig    := GVL_Mech.drvPress[0].MbWrExec;
            GVL_Mech.drvPress[0].MbWrDone := GVL_IO.iMbPr1Done AND GVL_Mech.drvPress[0].MbWrExec;
        2:  GVL_IO.qMbPr2Data[0] := GVL_Mech.drvPress[0].MbValH;
            GVL_IO.qMbPr2Data[1] := GVL_Mech.drvPress[0].MbValL;
            GVL_IO.qMbPr2Trig    := GVL_Mech.drvPress[0].MbWrExec;
            GVL_Mech.drvPress[0].MbWrDone := GVL_IO.iMbPr2Done AND GVL_Mech.drvPress[0].MbWrExec;
    END_CASE
    GVL_Mech.drvPress[0].MbWrErr :=
        (GVL_IO.iMbPrErr <> 0) AND GVL_Mech.drvPress[0].MbWrExec;
    // homing channel (FC06: 0x0020 -> 0x6002) + cyclic status word (0x1003)
    GVL_IO.qMbPrHomeData := 16#0020;
    GVL_IO.qMbPrHomeTrig := GVL_Mech.drvPress[0].MbHomeExec;
    GVL_Mech.drvPress[0].MbHomeDone :=
        GVL_IO.iMbPrHomeDone AND GVL_Mech.drvPress[0].MbHomeExec;
    GVL_Mech.drvPress[0].iStatusWord := GVL_IO.iMbPrStatus;
    // jog channel (FC06: 0x4001/0x4002 -> 0x1801)
    GVL_IO.qMbPrJogData := GVL_Mech.drvPress[0].MbJogVal;
    GVL_IO.qMbPrJogTrig := GVL_Mech.drvPress[0].MbJogExec;
    GVL_Mech.drvPress[0].MbJogDone :=
        GVL_IO.iMbPrJogDone AND GVL_Mech.drvPress[0].MbJogExec;
END_IF

// ---- pneumatics ----
GVL_Mech.fbDoorFridgeSide(Sim := GVL_Cfg.SIM_MODE, CycleMs := GVL_Cfg.T_APP_MS,
    iExtended := GVL_IO.iDoorFrSide_Op, iRetracted := GVL_IO.iDoorFrSide_Cl);
GVL_Mech.fbDoorChamber(Sim := GVL_Cfg.SIM_MODE, CycleMs := GVL_Cfg.T_APP_MS,
    iExtended := GVL_IO.iDoorChamber_Op, iRetracted := GVL_IO.iDoorChamber_Cl);
GVL_Mech.fbDoorFridgeFront(Sim := GVL_Cfg.SIM_MODE, CycleMs := GVL_Cfg.T_APP_MS,
    iExtended := GVL_IO.iDoorFrFront_Op, iRetracted := GVL_IO.iDoorFrFront_Cl);
GVL_Mech.fbPinGriddle(Sim := GVL_Cfg.SIM_MODE, CycleMs := GVL_Cfg.T_APP_MS,
    iExtended := GVL_IO.iPinGriddle_Ext, iRetracted := GVL_IO.iPinGriddle_Ret);
GVL_Mech.fbPinFridge(Sim := GVL_Cfg.SIM_MODE, CycleMs := GVL_Cfg.T_APP_MS,
    iExtended := GVL_IO.iPinFridge_Ext, iRetracted := GVL_IO.iPinFridge_Ret);
GVL_Mech.fbPneuGrip(Sim := GVL_Cfg.SIM_MODE, CycleMs := GVL_Cfg.T_APP_MS,
    iExtended := GVL_IO.iGripAcquired, iRetracted := NOT GVL_IO.iGripAcquired);
IF NOT GVL_Cfg.SIM_MODE THEN
    GVL_IO.qDoorFridgeSide  := GVL_Mech.fbDoorFridgeSide.qValve;
    GVL_IO.qDoorChamber     := GVL_Mech.fbDoorChamber.qValve;
    GVL_IO.qDoorFridgeFront := GVL_Mech.fbDoorFridgeFront.qValve;
    GVL_IO.qPinGriddle      := GVL_Mech.fbPinGriddle.qValve;
    GVL_IO.qPinFridge       := GVL_Mech.fbPinFridge.qValve;
    GVL_IO.qGripper         := GVL_Mech.fbPneuGrip.qValve;
END_IF

// ---- airlock ----
GVL_Mech.fbAirlock(
    Enable := GVL_Sts.enMotion, Abort := GVL_Sts.abortAll,
    DoorFridge := GVL_Mech.fbDoorFridgeSide,
    DoorChamber := GVL_Mech.fbDoorChamber);

// ---- carousels ----
GVL_Mech.vfdGriddle.Sim := GVL_Cfg.SIM_MODE;  GVL_Mech.vfdGriddle.CycleMs := GVL_Cfg.T_APP_MS;
GVL_Mech.vfdGriddle.iEnc := GVL_IO.diGridCarEnc;
GVL_Mech.vfdGriddle.iHomeProx := GVL_IO.iGridCarHome;
GVL_Mech.vfdFridge.Sim := GVL_Cfg.SIM_MODE;   GVL_Mech.vfdFridge.CycleMs := GVL_Cfg.T_APP_MS;
GVL_Mech.vfdFridge.iEnc := GVL_IO.diFrCarEnc;
GVL_Mech.vfdFridge.iHomeProx := GVL_IO.iFrCarHome;

GVL_Mech.fbGridCar(
    Enable := GVL_Sts.enMotion, Abort := GVL_Sts.abortAll,
    Vfd := GVL_Mech.vfdGriddle, Pin := GVL_Mech.fbPinGriddle);
GVL_Mech.fbFridgeCar(
    Enable := GVL_Sts.enMotion, Abort := GVL_Sts.abortAll,
    Vfd := GVL_Mech.vfdFridge, Pin := GVL_Mech.fbPinFridge);
GVL_Mech.vfdGriddle();
GVL_Mech.vfdFridge();
IF NOT GVL_Cfg.SIM_MODE THEN
    GVL_IO.qGridCarFwd := GVL_Mech.vfdGriddle.qFwd;
    GVL_IO.qGridCarRev := GVL_Mech.vfdGriddle.qRev;
    GVL_IO.wGridCarSpeed := GVL_Mech.vfdGriddle.qSpeed;
    GVL_IO.qFrCarFwd := GVL_Mech.vfdFridge.qFwd;
    GVL_IO.qFrCarRev := GVL_Mech.vfdFridge.qRev;
    GVL_IO.wFrCarSpeed := GVL_Mech.vfdFridge.qSpeed;
END_IF
GVL_Sts.carGridStation := GVL_Mech.fbGridCar.ActStation;
GVL_Sts.carFridgeFace  := GVL_Mech.fbFridgeCar.ActFace;

END_PROGRAM

// Device/Application/04_L3_Coordination/PRG_JobExec
(* ============================================================
   PRG_JobExec — executes Gateway primitives (T_App, after
   Supervisor). Enforces ORDER SAFETY only; scheduling policy is
   the Gateway's. Autonomous behavior: if a cook completes and the
   Gateway is silent (or no command pending), scrape locally —
   patties never burn waiting for a dead PC.
   In testMode this program idles (PRG_Test has authority).
   Primitive sub-sequences use numbered CASE states:
     100+ FETCH_TRAY   200+ LOAD_GRIDDLE   300+ SCRAPE
     400+ RETURN_TRAY
   ============================================================ *)
PROGRAM PRG_JobExec
VAR
    iSt        : INT;
    g         : INT;       // target griddle
    item      : UINT;
    count     : INT;
    level, face : INT;
    i         : INT;       // patty loop index
    trayIdx   : INT;
    batchSeq  : UDINT;
    autoScrape: BOOL;
    rotPerm   : BOOL;
    tonGw     : TON;
    tonStep   : TON;
    scrapeStroke : INT;
END_VAR


// ---- Gateway liveness ----
tonGw(IN := TRUE, PT := T#10S);   // re-armed by comms on heartbeat change
IF GVL_Cmd.gwAlive THEN tonGw(IN := FALSE); tonGw(IN := TRUE); END_IF
GVL_Sts.gwSilent := NOT GVL_Cmd.gwAlive;

// ---- rotation permissive for the griddle carousel ----
rotPerm := TRUE;
FOR i := 0 TO 3 DO
    // presses may rotate while HOLDING (they travel with the disc) but
    // never mid-motion
    IF GVL_Mech.fbPress[i].Busy THEN rotPerm := FALSE; END_IF
END_FOR
IF NOT GVL_Mech.fbGantry.Parked  THEN rotPerm := FALSE; END_IF
IF NOT GVL_Mech.fbScraper.Parked THEN rotPerm := FALSE; END_IF
GVL_Mech.fbGridCar.RotatePermissive := rotPerm;

// ---- tracker body (always runs) ----
GVL_Mech.fbTracker(Sim := GVL_Cfg.SIM_MODE);
GVL_Sts.aGriddle := GVL_Mech.fbTracker.aG;

// clear tracker command pulses after body call
GVL_Mech.fbTracker.SetLoading  := FALSE;
GVL_Mech.fbTracker.StartCook   := FALSE;
GVL_Mech.fbTracker.ScrapeStart := FALSE;
GVL_Mech.fbTracker.ScrapeDone  := FALSE;

IF GVL_Cmd.testMode THEN RETURN; END_IF
IF GVL_Sts.mode <> E_MachMode.RUN THEN
    IF iSt <> 0 THEN iSt := 0; END_IF   // mode fell out mid-primitive: mechanisms abort via Supervisor
    RETURN;
END_IF

tonStep(IN := iSt <> 0, PT := T#300S);
IF tonStep.Q AND (iSt <> 0) THEN
    GVL_Cmd.gwAck.error := TRUE;
    GVL_Cmd.gwAck.errorId := F_Err(GVL_Cfg.SS_JOBEXEC, GVL_Cfg.ERR_TIMEOUT);
    GVL_Cmd.gwAck.busy := FALSE; GVL_Cmd.gwPending := FALSE;
    iSt := 0;
END_IF

CASE iSt OF
    0: // ---- dispatch ----
        autoScrape := FALSE;
        IF GVL_Cmd.gwPending THEN
            IF GVL_Cmd.gwCmd.code = GVL_Cfg.CMD_FETCH_TRAY THEN
                item := TO_UINT(GVL_Cmd.gwCmd.p1); level := TO_INT(GVL_Cmd.gwCmd.p2); face := TO_INT(GVL_Cmd.gwCmd.p3);
                iSt := 100;
            ELSIF GVL_Cmd.gwCmd.code = GVL_Cfg.CMD_LOAD_GRIDDLE THEN
                g := TO_INT(GVL_Cmd.gwCmd.p1); count := TO_INT(GVL_Cmd.gwCmd.p2); item := TO_UINT(GVL_Cmd.gwCmd.p3);
                IF (g < 0) OR (g > 3) OR (count < 1) OR (count > GVL_Cfg.PATTIES_PER_GRIDDLE)
                   OR (GVL_Sts.aGriddle[g].state <> TO_UINT(E_GriddleState.EMPTY))
                   OR (NOT GVL_Sts.tray.inChamber) OR (GVL_Sts.tray.remaining < count) THEN
                    GVL_Cmd.gwAck.error := TRUE;
                    GVL_Cmd.gwAck.errorId := F_Err(GVL_Cfg.SS_JOBEXEC, GVL_Cfg.ERR_BAD_CMD);
                    GVL_Cmd.gwAck.busy := FALSE; GVL_Cmd.gwPending := FALSE;
                ELSE
                    iSt := 200;
                END_IF
            ELSIF GVL_Cmd.gwCmd.code = GVL_Cfg.CMD_SCRAPE THEN
                g := TO_INT(GVL_Cmd.gwCmd.p1);
                iSt := 300;
            ELSIF GVL_Cmd.gwCmd.code = GVL_Cfg.CMD_RETURN_TRAY THEN
                level := TO_INT(GVL_Cmd.gwCmd.p1); face := TO_INT(GVL_Cmd.gwCmd.p2);
                iSt := 400;
            ELSIF GVL_Cmd.gwCmd.code = GVL_Cfg.CMD_CLEAN_MODE THEN
                GVL_Cmd.reqClean := TRUE;
                GVL_Cmd.gwAck.done := TRUE; GVL_Cmd.gwAck.busy := FALSE; GVL_Cmd.gwPending := FALSE;
            ELSIF GVL_Cmd.gwCmd.code = GVL_Cfg.CMD_ABORT THEN
                GVL_Cmd.reqStop := TRUE;
                GVL_Cmd.gwAck.done := TRUE; GVL_Cmd.gwAck.busy := FALSE; GVL_Cmd.gwPending := FALSE;
            ELSE
                GVL_Cmd.gwAck.error := TRUE;
                GVL_Cmd.gwAck.errorId := F_Err(GVL_Cfg.SS_JOBEXEC, GVL_Cfg.ERR_BAD_CMD);
                GVL_Cmd.gwAck.busy := FALSE; GVL_Cmd.gwPending := FALSE;
            END_IF
        ELSIF GVL_Mech.fbTracker.ScrapeDue AND GVL_Sts.gwSilent THEN
            // AUTONOMOUS FINISH: gateway dead, cook done -> scrape locally
            g := GVL_Mech.fbTracker.ScrapeDueG;
            autoScrape := TRUE;
            iSt := 300;
        END_IF

    // ================= FETCH_TRAY =================
    100: // rotate fridge column to face (fork must be retracted/parked)
        GVL_Mech.fbFridgeCar.Permissive := NOT GVL_Mech.fbFork.Busy;
        GVL_Mech.fbFridgeCar.TargetFace := face;
        GVL_Mech.fbFridgeCar.GotoExec := TRUE;
        iSt := 101;
    101:
        IF GVL_Mech.fbFridgeCar.Done OR (GVL_Mech.fbFridgeCar.ActFace = face) THEN
            GVL_Mech.fbFridgeCar.GotoExec := FALSE; iSt := 102;
        ELSIF GVL_Mech.fbFridgeCar.Error THEN iSt := 900;
        END_IF
    102: // open fridge-side gate
        GVL_Mech.fbAirlock.ReqFridgeOpen := TRUE;
        IF GVL_Mech.fbAirlock.FridgeOpen THEN iSt := 103; END_IF
        IF GVL_Mech.fbAirlock.Error THEN iSt := 900; END_IF
    103: // fork fetch
        GVL_Mech.fbFork.Cmd.code := GVL_Cfg.MCMD_FETCH;
        GVL_Mech.fbFork.Cmd.p1 := TO_LREAL(level);
        GVL_Mech.fbFork.CmdExec := TRUE;
        iSt := 104;
    104:
        IF GVL_Mech.fbFork.Done AND GVL_Mech.fbFork.TrayHeld THEN
            GVL_Mech.fbFork.CmdExec := FALSE; iSt := 105;
        ELSIF GVL_Mech.fbFork.Error THEN
            GVL_Mech.fbFork.CmdExec := FALSE; iSt := 900;
        END_IF
    105: // close gate; publish tray info
        GVL_Mech.fbAirlock.ReqFridgeOpen := FALSE;
        IF GVL_Mech.fbAirlock.ChamberSealed THEN
            GVL_Sts.tray.item := item;
            GVL_Sts.tray.remaining := GVL_Cfg.PATTIES_PER_TRAY;
            GVL_Sts.tray.level := level; GVL_Sts.tray.face := face;
            GVL_Sts.tray.inChamber := TRUE;
            iSt := 990;
        END_IF

    // ================= LOAD_GRIDDLE =================
    200: // bring griddle g to load station
        GVL_Mech.fbTracker.SetLoading := TRUE; GVL_Mech.fbTracker.GIdxA := g;
        GVL_Mech.fbGridCar.TargetStation := g;
        GVL_Mech.fbGridCar.GotoExec := TRUE;
        iSt := 201;
    201:
        IF GVL_Mech.fbGridCar.Done OR (GVL_Mech.fbGridCar.ActStation = g) THEN
            GVL_Mech.fbGridCar.GotoExec := FALSE; iSt := 202;
        ELSIF GVL_Mech.fbGridCar.Error THEN iSt := 900;
        END_IF
    202: // open chamber gate (fridge side must be sealed)
        GVL_Mech.fbAirlock.ReqChamberOpen := TRUE;
        IF GVL_Mech.fbAirlock.ChamberOpen THEN i := 0; iSt := 210; END_IF
        IF GVL_Mech.fbAirlock.Error THEN iSt := 900; END_IF
    210: // pick patty i from tray
        trayIdx := GVL_Cfg.PATTIES_PER_TRAY - GVL_Sts.tray.remaining;
        GVL_Mech.fbGantry.Cmd.code := GVL_Cfg.MCMD_PICK;
        GVL_Mech.fbGantry.Cmd.p1 := TO_LREAL(trayIdx);
        GVL_Mech.fbGantry.CmdExec := TRUE;
        iSt := 211;
    211:
        IF GVL_Mech.fbGantry.Done THEN
            GVL_Mech.fbGantry.CmdExec := FALSE; iSt := 212;
        ELSIF GVL_Mech.fbGantry.Error THEN
            GVL_Mech.fbGantry.CmdExec := FALSE; iSt := 900;
        END_IF
    212: // place on griddle slot i
        GVL_Mech.fbGantry.Cmd.code := GVL_Cfg.MCMD_PLACE;
        GVL_Mech.fbGantry.Cmd.p1 := TO_LREAL(i);
        GVL_Mech.fbGantry.CmdExec := TRUE;
        iSt := 213;
    213:
        IF GVL_Mech.fbGantry.Done THEN
            GVL_Mech.fbGantry.CmdExec := FALSE;
            GVL_Sts.pattyOnGriddle[g, i] := TRUE;
            GVL_Sts.tray.remaining := GVL_Sts.tray.remaining - 1;
            i := i + 1;
            IF i >= count THEN iSt := 220; ELSE iSt := 210; END_IF
        ELSIF GVL_Mech.fbGantry.Error THEN
            GVL_Mech.fbGantry.CmdExec := FALSE; iSt := 900;
        END_IF
    220: // park gantry, close chamber
        GVL_Mech.fbGantry.Cmd.code := GVL_Cfg.MCMD_PARK;
        GVL_Mech.fbGantry.CmdExec := TRUE;
        iSt := 221;
    221:
        IF GVL_Mech.fbGantry.Done THEN
            GVL_Mech.fbGantry.CmdExec := FALSE;
            GVL_Mech.fbAirlock.ReqChamberOpen := FALSE;
            iSt := 222;
        ELSIF GVL_Mech.fbGantry.Error THEN
            GVL_Mech.fbGantry.CmdExec := FALSE; iSt := 900;
        END_IF
    222:
        IF GVL_Mech.fbAirlock.ChamberSealed THEN iSt := 230; END_IF
    230: // run press profile + start cook clock
        GVL_Mech.fbPress[g].Recipe := GVL_Par.aRecipe[item];
        GVL_Mech.fbPress[g].Cmd.code := GVL_Cfg.MCMD_PROFILE;
        GVL_Mech.fbPress[g].CmdExec := TRUE;
        iSt := 231;
    231:
        IF GVL_Mech.fbPress[g].Holding THEN
            GVL_Mech.fbPress[g].CmdExec := FALSE;
            batchSeq := batchSeq + 1;
            GVL_Mech.fbTracker.StartCook := TRUE;
            GVL_Mech.fbTracker.GIdxB := g;
            GVL_Mech.fbTracker.ItemB := item;
            GVL_Mech.fbTracker.CountB := count;
            GVL_Mech.fbTracker.BatchB := batchSeq;
            iSt := 990;
        ELSIF GVL_Mech.fbPress[g].Error THEN
            GVL_Mech.fbPress[g].CmdExec := FALSE; iSt := 900;
        END_IF

    // ================= SCRAPE =================
    300: // open press g first
        GVL_Mech.fbTracker.ScrapeStart := TRUE; GVL_Mech.fbTracker.GIdxC := g;
        GVL_Mech.fbPress[g].Cmd.code := GVL_Cfg.MCMD_OPEN;
        GVL_Mech.fbPress[g].CmdExec := TRUE;
        iSt := 301;
    301:
        IF GVL_Mech.fbPress[g].IsOpen THEN
            GVL_Mech.fbPress[g].CmdExec := FALSE; iSt := 302;
        ELSIF GVL_Mech.fbPress[g].Error THEN
            GVL_Mech.fbPress[g].CmdExec := FALSE; iSt := 900;
        END_IF
    302: // rotate griddle g to scrape station
        GVL_Mech.fbGridCar.TargetStation := (g + 2) MOD 4;
        GVL_Mech.fbGridCar.GotoExec := TRUE;
        iSt := 303;
    303:
        IF (GVL_Mech.fbGridCar.Done OR (GVL_Mech.fbGridCar.ActStation = (g + 2) MOD 4))
           AND NOT GVL_Mech.fbGridCar.Busy THEN   // arrival can be reported while still settling
            GVL_Mech.fbGridCar.GotoExec := FALSE;
            scrapeStroke := 0; iSt := 310;
        ELSIF GVL_Mech.fbGridCar.Error THEN iSt := 900;
        END_IF
    310: // sweep strokes — only command when the interlock is actually satisfied
        GVL_Mech.fbScraper.InterlockOk := GVL_Mech.fbPress[g].IsOpen AND NOT GVL_Mech.fbGridCar.Busy;
        IF GVL_Mech.fbScraper.InterlockOk THEN
            GVL_Mech.fbScraper.Cmd.code := GVL_Cfg.MCMD_SWEEP;
            GVL_Mech.fbScraper.Cmd.p1 := TO_LREAL(scrapeStroke);
            GVL_Mech.fbScraper.CmdExec := TRUE;
            iSt := 311;
        END_IF
    311:
        IF GVL_Mech.fbScraper.Done THEN
            GVL_Mech.fbScraper.CmdExec := FALSE;
            scrapeStroke := scrapeStroke + 1;
            IF scrapeStroke >= GVL_Cfg.SC_STROKES THEN iSt := 320; ELSE iSt := 310; END_IF
        ELSIF GVL_Mech.fbScraper.Error THEN
            GVL_Mech.fbScraper.CmdExec := FALSE; iSt := 900;
        END_IF
    320: // park scraper, finish batch bookkeeping
        GVL_Mech.fbScraper.Cmd.code := GVL_Cfg.MCMD_PARK;
        GVL_Mech.fbScraper.CmdExec := TRUE;
        iSt := 321;
    321:
        IF GVL_Mech.fbScraper.Done THEN
            GVL_Mech.fbScraper.CmdExec := FALSE;
            FOR i := 0 TO 5 DO GVL_Sts.pattyOnGriddle[g, i] := FALSE; END_FOR
            GVL_Mech.fbTracker.ScrapeDone := TRUE; GVL_Mech.fbTracker.GIdxD := g;
            iSt := 990;
        ELSIF GVL_Mech.fbScraper.Error THEN
            GVL_Mech.fbScraper.CmdExec := FALSE; iSt := 900;
        END_IF

    // ================= RETURN_TRAY =================
    400:
        GVL_Mech.fbAirlock.ReqFridgeOpen := TRUE;
        IF GVL_Mech.fbAirlock.FridgeOpen THEN iSt := 401; END_IF
        IF GVL_Mech.fbAirlock.Error THEN iSt := 900; END_IF
    401:
        GVL_Mech.fbFork.Cmd.code := GVL_Cfg.MCMD_RETURN;
        GVL_Mech.fbFork.Cmd.p1 := TO_LREAL(level);
        GVL_Mech.fbFork.CmdExec := TRUE;
        iSt := 402;
    402:
        IF GVL_Mech.fbFork.Done THEN
            GVL_Mech.fbFork.CmdExec := FALSE;
            GVL_Mech.fbAirlock.ReqFridgeOpen := FALSE;
            GVL_Sts.tray.inChamber := FALSE;
            iSt := 403;
        ELSIF GVL_Mech.fbFork.Error THEN
            GVL_Mech.fbFork.CmdExec := FALSE; iSt := 900;
        END_IF
    403:
        IF GVL_Mech.fbAirlock.ChamberSealed THEN iSt := 990; END_IF

    // ================= exits =================
    900: // primitive failed
        IF NOT autoScrape THEN
            GVL_Cmd.gwAck.error := TRUE;
            GVL_Cmd.gwAck.errorId := F_Err(GVL_Cfg.SS_JOBEXEC, GVL_Cfg.ERR_DRIVE);
            GVL_Cmd.gwAck.busy := FALSE; GVL_Cmd.gwPending := FALSE;
        END_IF
        iSt := 0;
    990: // primitive done
        IF NOT autoScrape THEN
            GVL_Cmd.gwAck.done := TRUE;
            GVL_Cmd.gwAck.busy := FALSE; GVL_Cmd.gwPending := FALSE;
        END_IF
        iSt := 0;
END_CASE

END_PROGRAM

// Device/Application/02_L1_Drivers/F_Err
(* ===== FUNCTION F_Err : UDINT =====
   ErrorID encoding: (subsystem << 16) OR code *)
FUNCTION F_Err : UDINT
VAR_INPUT
    ss   : UINT;
    code : UINT;
END_VAR

F_Err := SHL(TO_UDINT(ss), 16) OR TO_UDINT(code);

END_FUNCTION

// Device/Application/06_Wiring_Sim_Test/PRG_Test
(* ============================================================
   PRG_Test — automated regression suite (T_App, after JobExec).
   Start: set GVL_Cmd.testStart := TRUE (rising edge) once mode
   has reached READY. Results:
     aResult[n] : 0=pending 1=PASS 2=FAIL   (n = 1..10)
     aFailCode[n] : diagnostic (step*1000 or ErrorID low word)
     PassCount / suiteDone
   TC list:
     1  boot->READY + allHomed          6  griddle carousel 1,3,0
     2  IK table (24 pick + 6 place)    7  fork fetch/return L5
     3  heat AtSet + fridge + stagger   8  gantry pick/place/park
     4  airlock mutual exclusion        9  full cycle via Gateway regs
     5  press smash->hold->open        10  fault inject + recovery x2
   ============================================================ *)
PROGRAM PRG_Test
VAR
    aResult   : ARRAY[1..10] OF INT;
    aFailCode : ARRAY[1..10] OF UDINT;
    PassCount : INT;
    suiteDone : BOOL;
    running   : BOOL;
    tc        : INT;        // current test case
    stp       : INT;        // step within test case
    rtStart   : R_TRIG;
    tonG      : TON;        // per-step guard timer
    ptCur     : TIME;
    i, k      : INT;
    // TC2 locals
    px, py    : LREAL;
    xr, yr    : LREAL;
    thR       : LREAL;
    ikFail    : BOOL;
    // TC3 locals
    nRamp     : INT;
    stagViol  : BOOL;
    // TC9 locals
    testSeq   : UINT;
    hbCnt     : UINT;
    hbDiv     : INT;
    haccp0    : UDINT;
    holdCnt   : INT;
    PI_       : LREAL := 3.14159265358979;
END_VAR

rtStart(CLK := GVL_Cmd.testStart);
IF rtStart.Q AND NOT running THEN
    running := TRUE; suiteDone := FALSE;
    FOR i := 1 TO 10 DO aResult[i] := 0; aFailCode[i] := 0; END_FOR
    PassCount := 0;
    tc := 1; stp := 0;
END_IF
IF NOT running THEN RETURN; END_IF

// keep simulated gateway heartbeat alive during the whole suite
hbDiv := hbDiv + 1;
IF hbDiv >= 25 THEN   // every 500 ms
    hbDiv := 0; hbCnt := hbCnt + 1;
    GVL_Cmd.mbCmdRegs[9] := hbCnt;
END_IF

// per-step guard
tonG(IN := TRUE, PT := ptCur);

CASE tc OF
// ================= TC1: boot -> READY =================
1:
    CASE stp OF
        0: ptCur := T#90S; tonG(IN := FALSE); stp := 1;
        1:
            IF (GVL_Sts.mode = E_MachMode.READY) AND GVL_Sts.allHomed THEN
                aResult[1] := 1; tc := 2; stp := 0;
            ELSIF tonG.Q THEN
                aResult[1] := 2; aFailCode[1] := TO_UDINT(TO_UINT(GVL_Sts.mode));
                tc := 2; stp := 0;
            END_IF
    END_CASE

// ================= TC2: IK table =================
2:
    ikFail := FALSE;
    FOR i := 0 TO GVL_Cfg.PATTIES_PER_TRAY - 1 DO
        px := GVL_Cfg.PICK_BASE_X + TO_LREAL(i MOD GVL_Cfg.TRAY_COLS) * GVL_Cfg.PICK_SPACING_X;
        py := GVL_Cfg.PICK_BASE_Y + TO_LREAL(i / GVL_Cfg.TRAY_COLS) * GVL_Cfg.PICK_SPACING_Y;
        GVL_Mech.fbIK(xCart := px, yCart := py);
        IF NOT GVL_Mech.fbIK.Reachable THEN ikFail := TRUE; aFailCode[2] := TO_UDINT(TO_UINT(i)); END_IF
        thR := GVL_Mech.fbIK.thetaDeg * PI_ / 180.0;
        xr := GVL_Mech.fbIK.xLin + GVL_Cfg.ARM_LEN * COS(thR);
        yr := GVL_Cfg.ARM_LEN * SIN(thR);
        IF (ABS(xr - px) > 0.01) OR (ABS(yr - py) > 0.01) THEN
            ikFail := TRUE; aFailCode[2] := 1000 + TO_UDINT(TO_UINT(i));
        END_IF
    END_FOR
    FOR i := 0 TO GVL_Cfg.PATTIES_PER_GRIDDLE - 1 DO
        px := GVL_Cfg.PLACE_BASE_X + TO_LREAL(i MOD GVL_Cfg.PLACE_COLS) * GVL_Cfg.PLACE_SPC_X;
        py := GVL_Cfg.PLACE_BASE_Y + TO_LREAL(i / GVL_Cfg.PLACE_COLS) * GVL_Cfg.PLACE_SPC_Y;
        GVL_Mech.fbIK(xCart := px, yCart := py);
        IF NOT GVL_Mech.fbIK.Reachable THEN ikFail := TRUE; aFailCode[2] := 2000 + TO_UDINT(TO_UINT(i)); END_IF
    END_FOR
    IF ikFail THEN aResult[2] := 2; ELSE aResult[2] := 1; END_IF
    tc := 3; stp := 0;

// ================= TC3: heat + fridge + stagger =================
3:
    CASE stp OF
        0: ptCur := T#240S; tonG(IN := FALSE); stagViol := FALSE; stp := 1;
        1:
            // stagger monitor: count zones actively ramping WITH token
            nRamp := 0;
            FOR i := 0 TO 7 DO
                IF GVL_Mech.fbHeatBank.Token[i]
                   AND ((GVL_Sts.aHeat[i].setC - GVL_Sts.aHeat[i].actC) > 20.0) THEN
                    nRamp := nRamp + 1;
                END_IF
            END_FOR
            IF nRamp > GVL_Cfg.HEAT_MAX_STAGGER THEN stagViol := TRUE; END_IF
            IF GVL_Sts.heatAtSet AND GVL_Sts.fridgeAtSet THEN
                IF stagViol THEN aResult[3] := 2; aFailCode[3] := 1;
                ELSE aResult[3] := 1; END_IF
                tc := 4; stp := 0;
            ELSIF tonG.Q THEN
                aResult[3] := 2; aFailCode[3] := 2;
                tc := 4; stp := 0;
            END_IF
    END_CASE

// ================= TC4: airlock mutual exclusion =================
4:
    CASE stp OF
        0:
            ptCur := T#10S; tonG(IN := FALSE);
            GVL_Mech.fbAirlock.ReqFridgeOpen := TRUE;
            stp := 1;
        1:
            IF GVL_Mech.fbAirlock.FridgeOpen THEN
                GVL_Mech.fbAirlock.ReqChamberOpen := TRUE;  // request BOTH
                tonG(IN := FALSE); stp := 2;
            ELSIF tonG.Q THEN stp := 90; END_IF
        2: // hold both requests 2 s; invariant must hold
            IF GVL_Mech.fbAirlock.FridgeOpen AND GVL_Mech.fbAirlock.ChamberOpen THEN stp := 90; END_IF
            IF tonG.ET >= T#2S THEN
                GVL_Mech.fbAirlock.ReqFridgeOpen := FALSE;   // yield to chamber
                tonG(IN := FALSE); stp := 3;
            END_IF
        3:
            IF GVL_Mech.fbAirlock.FridgeOpen AND GVL_Mech.fbAirlock.ChamberOpen THEN stp := 90; END_IF
            IF GVL_Mech.fbAirlock.ChamberOpen THEN
                GVL_Mech.fbAirlock.ReqChamberOpen := FALSE;
                tonG(IN := FALSE); stp := 4;
            ELSIF tonG.Q THEN stp := 90; END_IF
        4:
            IF GVL_Mech.fbAirlock.ChamberSealed THEN
                aResult[4] := 1; tc := 5; stp := 0;
            ELSIF tonG.Q THEN stp := 90; END_IF
        90:
            GVL_Mech.fbAirlock.ReqFridgeOpen := FALSE;
            GVL_Mech.fbAirlock.ReqChamberOpen := FALSE;
            aResult[4] := 2; aFailCode[4] := TO_UDINT(TO_UINT(stp));
            tc := 5; stp := 0;
    END_CASE

// ================= TC5: press profile =================
5:
    CASE stp OF
        0:
            ptCur := T#20S; tonG(IN := FALSE);
            GVL_Mech.fbPress[0].Recipe := GVL_Par.aRecipe[1];   // BEEF
            GVL_Mech.fbPress[0].Cmd.code := GVL_Cfg.MCMD_PROFILE;
            GVL_Mech.fbPress[0].CmdExec := TRUE;
            stp := 1;
        1:
            IF GVL_Mech.fbPress[0].Holding THEN
                GVL_Mech.fbPress[0].CmdExec := FALSE;
                IF GVL_Mech.fbPress[0].DwellS < GVL_Par.aRecipe[1].smashDurS - 1.0 THEN
                    aFailCode[5] := 1; stp := 90;
                ELSE
                    GVL_Mech.fbPress[0].Cmd.code := GVL_Cfg.MCMD_OPEN;
                    tonG(IN := FALSE); stp := 12;   // one-scan gap: R_TRIG needs FALSE->TRUE across scans
                END_IF
            ELSIF GVL_Mech.fbPress[0].Error OR tonG.Q THEN
                GVL_Mech.fbPress[0].CmdExec := FALSE;
                aFailCode[5] := GVL_Mech.fbPress[0].ErrorID; stp := 90;
            END_IF
        12: // re-arm on a fresh scan
            GVL_Mech.fbPress[0].CmdExec := TRUE;
            stp := 2;
        2:
            IF GVL_Mech.fbPress[0].IsOpen THEN
                GVL_Mech.fbPress[0].CmdExec := FALSE;
                aResult[5] := 1; tc := 6; stp := 0;
            ELSIF GVL_Mech.fbPress[0].Error OR tonG.Q THEN
                GVL_Mech.fbPress[0].CmdExec := FALSE;
                aFailCode[5] := GVL_Mech.fbPress[0].ErrorID; stp := 90;
            END_IF
        90:
            aResult[5] := 2; tc := 6; stp := 0;
    END_CASE

// ================= TC6: griddle carousel =================
6:
    CASE stp OF
        0: // park gantry first so rotation permissive is TRUE
            ptCur := T#20S; tonG(IN := FALSE);
            GVL_Mech.fbGantry.Cmd.code := GVL_Cfg.MCMD_PARK;
            GVL_Mech.fbGantry.CmdExec := TRUE;
            stp := 1;
        1:
            IF GVL_Mech.fbGantry.Done AND GVL_Mech.fbGantry.Parked THEN
                GVL_Mech.fbGantry.CmdExec := FALSE; k := 0;
                tonG(IN := FALSE); stp := 2;
            ELSIF GVL_Mech.fbGantry.Error OR tonG.Q THEN
                GVL_Mech.fbGantry.CmdExec := FALSE;
                aFailCode[6] := GVL_Mech.fbGantry.ErrorID; stp := 90;
            END_IF
        2: // sequence of targets 1, 3, 0
            CASE k OF 0: i := 1; 1: i := 3; 2: i := 0; END_CASE
            GVL_Mech.fbGridCar.TargetStation := i;
            GVL_Mech.fbGridCar.GotoExec := TRUE;
            tonG(IN := FALSE); stp := 3;
        3:
            IF GVL_Mech.fbGridCar.Done AND (GVL_Mech.fbGridCar.ActStation = i) THEN
                GVL_Mech.fbGridCar.GotoExec := FALSE;
                k := k + 1;
                IF k >= 3 THEN aResult[6] := 1; tc := 7; stp := 0;
                ELSE stp := 2; END_IF
            ELSIF GVL_Mech.fbGridCar.Error OR tonG.Q THEN
                GVL_Mech.fbGridCar.GotoExec := FALSE;
                aFailCode[6] := GVL_Mech.fbGridCar.ErrorID; stp := 90;
            END_IF
        90:
            aResult[6] := 2; tc := 7; stp := 0;
    END_CASE

// ================= TC7: fork fetch / return =================
7:
    CASE stp OF
        0:
            ptCur := T#40S; tonG(IN := FALSE);
            GVL_Mech.fbFork.Cmd.code := GVL_Cfg.MCMD_FETCH;
            GVL_Mech.fbFork.Cmd.p1 := 5.0;
            GVL_Mech.fbFork.CmdExec := TRUE;
            stp := 1;
        1:
            IF GVL_Mech.fbFork.Done AND GVL_Mech.fbFork.TrayHeld THEN
                GVL_Mech.fbFork.CmdExec := FALSE;
                GVL_Mech.fbFork.Cmd.code := GVL_Cfg.MCMD_RETURN;
                GVL_Mech.fbFork.Cmd.p1 := 5.0;
                tonG(IN := FALSE); stp := 12;   // one-scan gap for a real edge
            ELSIF GVL_Mech.fbFork.Error OR tonG.Q THEN
                GVL_Mech.fbFork.CmdExec := FALSE;
                aFailCode[7] := GVL_Mech.fbFork.ErrorID; stp := 90;
            END_IF
        12: // re-arm on a fresh scan
            GVL_Mech.fbFork.CmdExec := TRUE;
            stp := 2;
        2:
            IF GVL_Mech.fbFork.Done AND NOT GVL_Mech.fbFork.TrayHeld THEN
                GVL_Mech.fbFork.CmdExec := FALSE;
                aResult[7] := 1; tc := 8; stp := 0;
            ELSIF GVL_Mech.fbFork.Error OR tonG.Q THEN
                GVL_Mech.fbFork.CmdExec := FALSE;
                aFailCode[7] := GVL_Mech.fbFork.ErrorID; stp := 90;
            END_IF
        90:
            aResult[7] := 2; tc := 8; stp := 0;
    END_CASE

// ================= TC8: gantry pick / place / park =================
8:
    CASE stp OF
        0:
            ptCur := T#30S; tonG(IN := FALSE);
            GVL_Mech.fbGantry.Cmd.code := GVL_Cfg.MCMD_PICK;
            GVL_Mech.fbGantry.Cmd.p1 := 0.0;
            GVL_Mech.fbGantry.CmdExec := TRUE;
            stp := 1;
        1:
            IF GVL_Mech.fbGantry.Done AND GVL_Mech.fbGripper.Holding THEN
                GVL_Mech.fbGantry.CmdExec := FALSE;
                GVL_Mech.fbGantry.Cmd.code := GVL_Cfg.MCMD_PLACE;
                GVL_Mech.fbGantry.Cmd.p1 := 0.0;
                tonG(IN := FALSE); stp := 12;   // one-scan gap for a real edge
            ELSIF GVL_Mech.fbGantry.Error OR tonG.Q THEN
                GVL_Mech.fbGantry.CmdExec := FALSE;
                aFailCode[8] := GVL_Mech.fbGantry.ErrorID; stp := 90;
            END_IF
        2:
            IF GVL_Mech.fbGantry.Done AND NOT GVL_Mech.fbGripper.Holding THEN
                GVL_Mech.fbGantry.CmdExec := FALSE;
                GVL_Mech.fbGantry.Cmd.code := GVL_Cfg.MCMD_PARK;
                tonG(IN := FALSE); stp := 13;   // one-scan gap for a real edge
            ELSIF GVL_Mech.fbGantry.Error OR tonG.Q THEN
                GVL_Mech.fbGantry.CmdExec := FALSE;
                aFailCode[8] := GVL_Mech.fbGantry.ErrorID; stp := 90;
            END_IF
        12: // re-arm PLACE on a fresh scan
            GVL_Mech.fbGantry.CmdExec := TRUE;
            stp := 2;
        13: // re-arm PARK on a fresh scan
            GVL_Mech.fbGantry.CmdExec := TRUE;
            stp := 3;
        3:
            IF GVL_Mech.fbGantry.Done AND GVL_Mech.fbGantry.Parked THEN
                GVL_Mech.fbGantry.CmdExec := FALSE;
                aResult[8] := 1; tc := 9; stp := 0;
            ELSIF GVL_Mech.fbGantry.Error OR tonG.Q THEN
                GVL_Mech.fbGantry.CmdExec := FALSE;
                aFailCode[8] := GVL_Mech.fbGantry.ErrorID; stp := 90;
            END_IF
        90:
            aResult[8] := 2; tc := 9; stp := 0;
    END_CASE

// ================= TC9: full cycle via Gateway registers =================
9:
    CASE stp OF
        0: // enter RUN through the real path — but first wait for thermal readiness
           // (fridge pulldown / heat-up gate READY->RUN; on a fast suite run they
           //  may not be satisfied yet)
            GVL_Cmd.testMode := FALSE;
            haccp0 := GVL_Sts.haccpCount;
            ptCur := T#300S; tonG(IN := FALSE); stp := 30;
        30:
            IF GVL_Sts.heatAtSet AND GVL_Sts.fridgeAtSet AND GVL_Sts.allHomed THEN
                GVL_Cmd.reqStart := TRUE; holdCnt := 0;
                ptCur := T#20S; tonG(IN := FALSE); stp := 1;
            ELSIF tonG.Q THEN aFailCode[9] := 30; stp := 90; END_IF
        1:
            holdCnt := holdCnt + 1;
            IF holdCnt > 5 THEN GVL_Cmd.reqStart := FALSE; END_IF
            IF holdCnt > 10 THEN GVL_Cmd.reqStart := TRUE; holdCnt := 0; END_IF  // retry edge (one-shot may be rejected)
            IF GVL_Sts.mode = E_MachMode.RUN THEN
                GVL_Cmd.reqStart := FALSE; stp := 2;
            ELSIF tonG.Q THEN aFailCode[9] := 1; stp := 90; END_IF
        2: // FETCH_TRAY item=1 level=3 face=0
            testSeq := testSeq + 1;
            GVL_Cmd.mbCmdRegs[0] := testSeq;
            GVL_Cmd.mbCmdRegs[1] := GVL_Cfg.CMD_FETCH_TRAY;
            GVL_Cmd.mbCmdRegs[2] := 1;  GVL_Cmd.mbCmdRegs[3] := 0;   // p1 item
            GVL_Cmd.mbCmdRegs[4] := 3;  GVL_Cmd.mbCmdRegs[5] := 0;   // p2 level
            GVL_Cmd.mbCmdRegs[6] := 0;  GVL_Cmd.mbCmdRegs[7] := 0;   // p3 face
            ptCur := T#60S; tonG(IN := FALSE); stp := 3;
        3:
            IF (GVL_Cmd.gwAck.seqEcho = testSeq) AND GVL_Cmd.gwAck.done THEN stp := 4;
            ELSIF (GVL_Cmd.gwAck.seqEcho = testSeq) AND GVL_Cmd.gwAck.error THEN
                aFailCode[9] := GVL_Cmd.gwAck.errorId; stp := 90;
            ELSIF tonG.Q THEN aFailCode[9] := 3; stp := 90; END_IF
        4: // LOAD_GRIDDLE g=0 count=2 item=1
            testSeq := testSeq + 1;
            GVL_Cmd.mbCmdRegs[0] := testSeq;
            GVL_Cmd.mbCmdRegs[1] := GVL_Cfg.CMD_LOAD_GRIDDLE;
            GVL_Cmd.mbCmdRegs[2] := 0;  GVL_Cmd.mbCmdRegs[3] := 0;
            GVL_Cmd.mbCmdRegs[4] := 2;  GVL_Cmd.mbCmdRegs[5] := 0;
            GVL_Cmd.mbCmdRegs[6] := 1;  GVL_Cmd.mbCmdRegs[7] := 0;
            ptCur := T#120S; tonG(IN := FALSE); stp := 5;
        5:
            IF (GVL_Cmd.gwAck.seqEcho = testSeq) AND GVL_Cmd.gwAck.done THEN stp := 6;
            ELSIF (GVL_Cmd.gwAck.seqEcho = testSeq) AND GVL_Cmd.gwAck.error THEN
                aFailCode[9] := GVL_Cmd.gwAck.errorId; stp := 90;
            ELSIF tonG.Q THEN aFailCode[9] := 5; stp := 90; END_IF
        6: // wait cook done (90 s scaled by 5 -> ~18 s real)
            ptCur := T#120S; tonG(IN := FALSE); stp := 7;
        7:
            IF GVL_Sts.aGriddle[0].state = TO_UINT(E_GriddleState.READY_TO_SCRAPE) THEN stp := 8;
            ELSIF tonG.Q THEN aFailCode[9] := 7; stp := 90; END_IF
        8: // SCRAPE g=0
            testSeq := testSeq + 1;
            GVL_Cmd.mbCmdRegs[0] := testSeq;
            GVL_Cmd.mbCmdRegs[1] := GVL_Cfg.CMD_SCRAPE;
            GVL_Cmd.mbCmdRegs[2] := 0;  GVL_Cmd.mbCmdRegs[3] := 0;
            GVL_Cmd.mbCmdRegs[4] := 0;  GVL_Cmd.mbCmdRegs[6] := 0;
            ptCur := T#90S; tonG(IN := FALSE); stp := 9;
        9:
            IF (GVL_Cmd.gwAck.seqEcho = testSeq) AND GVL_Cmd.gwAck.done THEN stp := 10;
            ELSIF (GVL_Cmd.gwAck.seqEcho = testSeq) AND GVL_Cmd.gwAck.error THEN
                aFailCode[9] := GVL_Cmd.gwAck.errorId; stp := 90;
            ELSIF tonG.Q THEN aFailCode[9] := 9; stp := 90; END_IF
        10: // RETURN_TRAY level=3 face=0
            testSeq := testSeq + 1;
            GVL_Cmd.mbCmdRegs[0] := testSeq;
            GVL_Cmd.mbCmdRegs[1] := GVL_Cfg.CMD_RETURN_TRAY;
            GVL_Cmd.mbCmdRegs[2] := 3;  GVL_Cmd.mbCmdRegs[3] := 0;
            GVL_Cmd.mbCmdRegs[4] := 0;  GVL_Cmd.mbCmdRegs[5] := 0;
            ptCur := T#60S; tonG(IN := FALSE); stp := 11;
        11:
            IF (GVL_Cmd.gwAck.seqEcho = testSeq) AND GVL_Cmd.gwAck.done THEN
                // HACCP record must exist and be clean
                IF (GVL_Sts.haccpCount = haccp0 + 1) AND (GVL_Sts.lastHaccp.result = 0) THEN
                    aResult[9] := 1;
                ELSE
                    aResult[9] := 2; aFailCode[9] := 11;
                END_IF
                GVL_Cmd.testMode := TRUE;
                tc := 10; stp := 0;
            ELSIF (GVL_Cmd.gwAck.seqEcho = testSeq) AND GVL_Cmd.gwAck.error THEN
                aFailCode[9] := GVL_Cmd.gwAck.errorId; stp := 90;
            ELSIF tonG.Q THEN aFailCode[9] := 12; stp := 90; END_IF
        90:
            GVL_Cmd.testMode := TRUE;
            aResult[9] := 2; tc := 10; stp := 0;
    END_CASE

// ================= TC10: fault injection + recovery =================
10:
    CASE stp OF
        0: // inject: unreachable gantry target (idx 99 -> y >> arm)
            ptCur := T#30S; tonG(IN := FALSE);
            GVL_Mech.fbGantry.Cmd.code := GVL_Cfg.MCMD_PLACE;
            GVL_Mech.fbGantry.Cmd.p1 := 99.0;
            GVL_Mech.fbGantry.CmdExec := FALSE;  // may be left TRUE by JobExec (TC9) — force an edge
            stp := 20;
        20: // arm on a fresh scan
            GVL_Mech.fbGantry.CmdExec := TRUE;
            stp := 1;
        1:
            IF GVL_Mech.fbGantry.Error THEN
                GVL_Mech.fbGantry.CmdExec := FALSE;
                IF (GVL_Mech.fbGantry.ErrorID AND 16#FFFF) <> TO_UDINT(GVL_Cfg.ERR_UNREACH) THEN
                    aFailCode[10] := GVL_Mech.fbGantry.ErrorID; stp := 90;
                ELSE
                    tonG(IN := FALSE); stp := 2;
                END_IF
            ELSIF tonG.Q THEN aFailCode[10] := 1; stp := 90; END_IF
        2: // system must fall to FAULT via alarm cascade
            IF GVL_Sts.mode = E_MachMode.FAULT THEN
                GVL_Cmd.reqAckAll := TRUE; holdCnt := 0;
                tonG(IN := FALSE); stp := 3;
            ELSIF tonG.Q THEN aFailCode[10] := 2; stp := 90; END_IF
        3:
            holdCnt := holdCnt + 1;
            IF holdCnt > 5 THEN
                GVL_Cmd.reqAckAll := FALSE;
                GVL_Cmd.reqReset := TRUE; holdCnt := 0;
                stp := 4;
            END_IF
        4:
            holdCnt := holdCnt + 1;
            IF holdCnt > 5 THEN GVL_Cmd.reqReset := FALSE; END_IF
            IF holdCnt > 10 THEN GVL_Cmd.reqReset := TRUE; holdCnt := 0; END_IF  // retry edge
            IF GVL_Sts.mode = E_MachMode.HOMING THEN
                GVL_Cmd.reqReset := FALSE;
                ptCur := T#90S; tonG(IN := FALSE); stp := 5;
            ELSIF tonG.Q THEN aFailCode[10] := 4; stp := 90; END_IF
        5:
            IF (GVL_Sts.mode = E_MachMode.READY) AND GVL_Sts.allHomed THEN
                tonG(IN := FALSE); stp := 6;
            ELSIF tonG.Q THEN aFailCode[10] := 5; stp := 90; END_IF
        6: // inject 2: scraper sweep with interlock FALSE
            GVL_Mech.fbScraper.InterlockOk := FALSE;
            GVL_Mech.fbScraper.Cmd.code := GVL_Cfg.MCMD_SWEEP;
            GVL_Mech.fbScraper.Cmd.p1 := 0.0;
            GVL_Mech.fbScraper.CmdExec := TRUE;
            ptCur := T#20S; tonG(IN := FALSE); stp := 7;
        7:
            IF GVL_Mech.fbScraper.Error THEN
                GVL_Mech.fbScraper.CmdExec := FALSE;
                IF (GVL_Mech.fbScraper.ErrorID AND 16#FFFF) <> TO_UDINT(GVL_Cfg.ERR_INTERLOCK) THEN
                    aFailCode[10] := GVL_Mech.fbScraper.ErrorID; stp := 90;
                ELSE
                    tonG(IN := FALSE); stp := 8;
                END_IF
            ELSIF tonG.Q THEN aFailCode[10] := 7; stp := 90; END_IF
        8: // recover again
            IF GVL_Sts.mode = E_MachMode.FAULT THEN
                GVL_Cmd.reqAckAll := TRUE; holdCnt := 0; stp := 9;
            ELSIF tonG.Q THEN aFailCode[10] := 8; stp := 90; END_IF
        9:
            holdCnt := holdCnt + 1;
            IF holdCnt > 5 THEN
                GVL_Cmd.reqAckAll := FALSE;
                GVL_Cmd.reqReset := TRUE; holdCnt := 0;
                ptCur := T#90S; tonG(IN := FALSE); stp := 11;
            END_IF
        11:
            holdCnt := holdCnt + 1;
            IF holdCnt > 5 THEN GVL_Cmd.reqReset := FALSE; END_IF
            IF (holdCnt > 10) AND (GVL_Sts.mode = E_MachMode.FAULT) THEN
                GVL_Cmd.reqReset := TRUE; holdCnt := 0;   // retry edge while still faulted
            END_IF
            IF (GVL_Sts.mode = E_MachMode.READY) AND GVL_Sts.allHomed THEN
                GVL_Cmd.reqReset := FALSE;
                aResult[10] := 1; stp := 99;
            ELSIF tonG.Q THEN aFailCode[10] := 11; stp := 90; END_IF
        90:
            GVL_Mech.fbGantry.CmdExec := FALSE;
            GVL_Mech.fbScraper.CmdExec := FALSE;
            aResult[10] := 2; stp := 99;
        99: // ---- suite complete ----
            PassCount := 0;
            FOR i := 1 TO 10 DO
                IF aResult[i] = 1 THEN PassCount := PassCount + 1; END_IF
            END_FOR
            suiteDone := TRUE; running := FALSE;
            GVL_Cmd.testStart := FALSE;
    END_CASE
END_CASE

END_PROGRAM

// Device/Application/06_Wiring_Sim_Test/PRG_Heating
(* ============================================================
   PRG_Heating — T_App body-call owner: 8 heaters + bank + fridge.
   Zone map: griddle g -> zones 2g (top), 2g+1 (bottom).
   Setpoint follows the active recipe of the griddle's item; empty
   griddles idle at the BEEF setpoint so they are ready to load.
   ============================================================ *)
PROGRAM PRG_Heating
VAR
    z, g : INT;
    itm  : UINT;
    setC : LREAL;
END_VAR

FOR z := 0 TO 7 DO
    g := z / 2;
    itm := GVL_Sts.aGriddle[g].item;
    IF itm = 0 THEN itm := 1; END_IF          // idle at BEEF setpoint
    setC := GVL_Par.aRecipe[itm].platenSetC;
    GVL_Mech.fbHeater[z].Sim := GVL_Cfg.SIM_MODE;
    GVL_Mech.fbHeater[z].ZoneId := z;
    GVL_Mech.fbHeater[z].CycleMs := GVL_Cfg.T_APP_MS;
    GVL_Mech.fbHeater[z].Enable := GVL_Sts.enProcess;
    GVL_Mech.fbHeater[z].SetC := setC;
    GVL_Mech.fbHeater[z].iTempRaw := GVL_IO.wPlatenTemp[z];
    GVL_Mech.fbHeater[z].StaggerToken := GVL_Mech.fbHeatBank.Token[z];
    GVL_Mech.fbHeater[z]();
    IF NOT GVL_Cfg.SIM_MODE THEN
        GVL_IO.qSsr[z] := GVL_Mech.fbHeater[z].qSsr;
    END_IF
    GVL_Sts.aHeat[z] := GVL_Mech.fbHeater[z].Zone;
END_FOR
GVL_Mech.fbHeatBank(Enable := GVL_Sts.enProcess, Heaters := GVL_Mech.fbHeater);

GVL_Mech.fbRefrig(
    Sim := GVL_Cfg.SIM_MODE,
    Enable := GVL_Sts.enProcess,
    iTempRaw := GVL_IO.wFridgeTemp,
    CycleMs := GVL_Cfg.T_APP_MS);
// (compressor output relay would be copied to GVL_IO here at migration)

END_PROGRAM

// Device/Application/06_Wiring_Sim_Test/PRG_Sim
(* ============================================================
   PRG_Sim — T_App. Plant models beyond what L1 drivers model
   internally. v1: reserved (axis/pneu/thermal/fridge models are
   inside their driver FBs; patty bookkeeping is in JobExec).
   Extend here for: patty-present optics model, condensation /
   door-open thermal coupling, disturbance injection.
   ============================================================ *)
PROGRAM PRG_Sim
VAR
END_VAR

;

END_PROGRAM

// Device/Application/05_L4_Comms/PRG_Alarms
(* ============================================================
   PRG_Alarms — central alarm manager (T_App, runs LAST).
   Raises on the RISING edge of each source Error (so an acked
   alarm doesn't re-raise from a still-latched source; sources
   clear their Error on the next command latch / axis reset).
   Class map (spec sec.13):
     MACHINE_STOP : fork brake/drive integrity
     ZONE_STOP    : axis/drive faults, pin mismatch, TC fault,
                    airlock violation, mechanism timeouts
     QUARANTINE   : fridge excursion, short-cook (via PRG_HACCP)
     INFO         : gateway silent
   ============================================================ *)
PROGRAM PRG_Alarms
VAR
    i, n : INT;
    worst: UINT;
    rtAck: R_TRIG;
    rtGw : R_TRIG;
    rtGan, rtScr, rtFrk, rtGC, rtFC, rtAir, rtExc : R_TRIG;
    rtPress  : ARRAY[0..3] OF R_TRIG;
    rtHeat   : ARRAY[0..7] OF R_TRIG;
END_VAR

// ---- collect (edge-raised) ----
rtFrk(CLK := GVL_Mech.fbFork.Error);
IF rtFrk.Q THEN
    IF SHR(GVL_Mech.fbFork.ErrorID, 16) = TO_UDINT(GVL_Cfg.SS_FORK_Z) THEN
        F_RaiseAlarm(GVL_Mech.fbFork.ErrorID, TO_UINT(E_FaultClass.MACHINE_STOP));
    ELSE
        F_RaiseAlarm(GVL_Mech.fbFork.ErrorID, TO_UINT(E_FaultClass.ZONE_STOP));
    END_IF
END_IF
rtGan(CLK := GVL_Mech.fbGantry.Error);
IF rtGan.Q THEN F_RaiseAlarm(GVL_Mech.fbGantry.ErrorID, TO_UINT(E_FaultClass.ZONE_STOP)); END_IF
rtScr(CLK := GVL_Mech.fbScraper.Error);
IF rtScr.Q THEN F_RaiseAlarm(GVL_Mech.fbScraper.ErrorID, TO_UINT(E_FaultClass.ZONE_STOP)); END_IF
rtGC(CLK := GVL_Mech.fbGridCar.Error);
IF rtGC.Q THEN F_RaiseAlarm(GVL_Mech.fbGridCar.ErrorID, TO_UINT(E_FaultClass.ZONE_STOP)); END_IF
rtFC(CLK := GVL_Mech.fbFridgeCar.Error);
IF rtFC.Q THEN F_RaiseAlarm(GVL_Mech.fbFridgeCar.ErrorID, TO_UINT(E_FaultClass.ZONE_STOP)); END_IF
rtAir(CLK := GVL_Mech.fbAirlock.Error);
IF rtAir.Q THEN F_RaiseAlarm(GVL_Mech.fbAirlock.ErrorID, TO_UINT(E_FaultClass.ZONE_STOP)); END_IF
FOR i := 0 TO 3 DO
    rtPress[i](CLK := GVL_Mech.fbPress[i].Error);
    IF rtPress[i].Q THEN
        F_RaiseAlarm(GVL_Mech.fbPress[i].ErrorID, TO_UINT(E_FaultClass.ZONE_STOP));
    END_IF
END_FOR
FOR i := 0 TO 7 DO
    rtHeat[i](CLK := GVL_Mech.fbHeater[i].Error);
    IF rtHeat[i].Q THEN
        F_RaiseAlarm(GVL_Mech.fbHeater[i].ErrorID, TO_UINT(E_FaultClass.ZONE_STOP));
    END_IF
END_FOR
rtExc(CLK := GVL_Mech.fbRefrig.Excursion);
IF rtExc.Q THEN
    F_RaiseAlarm(GVL_Mech.fbRefrig.ErrorID, TO_UINT(E_FaultClass.QUARANTINE));
END_IF
rtGw(CLK := GVL_Sts.gwSilent AND (GVL_Sts.mode = E_MachMode.RUN) AND NOT GVL_Cmd.testMode);
IF rtGw.Q THEN
    F_RaiseAlarm(F_Err(GVL_Cfg.SS_GWCOMMS, GVL_Cfg.ERR_TIMEOUT), TO_UINT(E_FaultClass.INFO));
END_IF

// ---- ack / clear ----
rtAck(CLK := GVL_Cmd.reqAckAll);
n := 0; worst := 0;
FOR i := 0 TO 63 DO
    IF GVL_Alm.aActive[i].active THEN
        IF rtAck.Q THEN GVL_Alm.aActive[i].acked := TRUE; END_IF
        IF GVL_Alm.aActive[i].acked THEN
            GVL_Alm.aActive[i].active := FALSE;
        ELSE
            n := n + 1;
            IF GVL_Alm.aActive[i].class > worst THEN worst := GVL_Alm.aActive[i].class; END_IF
        END_IF
    END_IF
END_FOR
GVL_Alm.nActive := n;
GVL_Alm.worstClass := worst;
GVL_Alm.reqZoneStop := worst >= TO_UINT(E_FaultClass.ZONE_STOP);
GVL_Alm.reqMachStop := worst >= TO_UINT(E_FaultClass.MACHINE_STOP);
GVL_Sts.activeAlarms := n;

END_PROGRAM

// Device/Application/02_L1_Drivers/F_RaiseAlarm
(* ===== FUNCTION F_RaiseAlarm : BOOL =====
   Latch an alarm into GVL_Alm (dedup by id). Returns TRUE if new. *)
FUNCTION F_RaiseAlarm : BOOL
VAR_INPUT
    id    : UDINT;
    class : UINT;   // E_FaultClass value
END_VAR
VAR
    i : INT;
END_VAR

F_RaiseAlarm := FALSE;
IF id = 0 THEN RETURN; END_IF
FOR i := 0 TO 63 DO
    IF GVL_Alm.aActive[i].active AND (GVL_Alm.aActive[i].id = id) THEN
        RETURN;                      // already active
    END_IF
END_FOR
FOR i := 0 TO 63 DO
    IF NOT GVL_Alm.aActive[i].active THEN
        GVL_Alm.aActive[i].id     := id;
        GVL_Alm.aActive[i].class  := class;
        GVL_Alm.aActive[i].tsS    := GVL_Sts.uptimeS;
        GVL_Alm.aActive[i].active := TRUE;
        GVL_Alm.aActive[i].acked  := FALSE;
        // history ring
        GVL_Alm.aHistory[GVL_Alm.histHead] := GVL_Alm.aActive[i];
        GVL_Alm.histHead := (GVL_Alm.histHead + 1) MOD 200;
        F_RaiseAlarm := TRUE;
        RETURN;
    END_IF
END_FOR

END_FUNCTION

// Device/Application/05_L4_Comms/PRG_HACCP
(* ============================================================
   PRG_HACCP — cook record collector (T_Comms). RETAIN ring of
   512 records (> one shift). Gateway currently reads the LATEST
   record snapshot from STS regs; full drain protocol via read
   pointer is a marked TODO for Gateway integration (M4).
   ============================================================ *)
PROGRAM PRG_HACCP
VAR RETAIN
    ring : ARRAY[0..511] OF ST_HaccpRec;
    head : INT;
END_VAR

IF GVL_Mech.fbTracker.NewHaccp AND NOT GVL_Mech.fbTracker.HaccpAck THEN
    ring[head] := GVL_Mech.fbTracker.HaccpRec;
    head := (head + 1) MOD 512;
    GVL_Sts.haccpCount := GVL_Sts.haccpCount + 1;
    GVL_Sts.lastHaccp := GVL_Mech.fbTracker.HaccpRec;
    IF GVL_Mech.fbTracker.HaccpRec.result = 1 THEN
        F_RaiseAlarm(F_Err(GVL_Cfg.SS_JOBEXEC, GVL_Cfg.ERR_SENSOR),
                     TO_UINT(E_FaultClass.QUARANTINE));
    END_IF
    GVL_Mech.fbTracker.HaccpAck := TRUE;       // tracker clears NewHaccp
ELSIF NOT GVL_Mech.fbTracker.NewHaccp THEN
    GVL_Mech.fbTracker.HaccpAck := FALSE;      // handshake complete, re-arm
END_IF

END_PROGRAM

// Device/Application/05_L4_Comms/PRG_GatewayComms
(* ============================================================
   PRG_GatewayComms — Modbus-TCP register map + seq/ack handshake
   (T_Comms, 100 ms). PLC is Modbus TCP slave; Gateway reads/writes
   the %MW images declared in GVL_Cmd.
   Register map (holding registers, 1 reg = 1 WORD):
     CMD  %MW0..9   : [0]=seq [1]=code [2..3]=p1 lo/hi [4..5]=p2
                      [6..7]=p3 [8]=p4(lo only) [9]=gwHeartbeat
     ACK  %MW10..15 : [10]=seqEcho [11]=flags(b0 busy b1 done b2 err)
                      [12..13]=errorId lo/hi [14]=plc heartbeat
     STS  %MW20..99 : see packing below
     PAR  %MW500..  : [500]=item [501]=cookTimeS*10 [502]=setC*10
                      [503]=applyToggle (change -> apply, READY only)
   ============================================================ *)
PROGRAM PRG_GatewayComms
VAR
    lastSeq     : UINT;
    lastHb      : UINT;
    hbAge       : INT;
    flags       : WORD;
    z, gIdx     : INT;
    parToggle   : WORD;
    lastParTog  : WORD;
    itemP       : INT;
    cookP, setP : LREAL;
END_VAR

// ---------- decode command ----------
GVL_Cmd.gwCmd.seq  := GVL_Cmd.mbCmdRegs[0];
GVL_Cmd.gwCmd.code := GVL_Cmd.mbCmdRegs[1];
GVL_Cmd.gwCmd.p1 := WORD_TO_DINT(GVL_Cmd.mbCmdRegs[2]) + SHL(WORD_TO_DINT(GVL_Cmd.mbCmdRegs[3]), 16);
GVL_Cmd.gwCmd.p2 := WORD_TO_DINT(GVL_Cmd.mbCmdRegs[4]) + SHL(WORD_TO_DINT(GVL_Cmd.mbCmdRegs[5]), 16);
GVL_Cmd.gwCmd.p3 := WORD_TO_DINT(GVL_Cmd.mbCmdRegs[6]) + SHL(WORD_TO_DINT(GVL_Cmd.mbCmdRegs[7]), 16);
GVL_Cmd.gwCmd.p4 := WORD_TO_DINT(GVL_Cmd.mbCmdRegs[8]);
GVL_Cmd.gwHeartbeatIn := GVL_Cmd.mbCmdRegs[9];

// ---------- gateway liveness (heartbeat must CHANGE) ----------
IF GVL_Cmd.gwHeartbeatIn <> lastHb THEN
    lastHb := GVL_Cmd.gwHeartbeatIn; hbAge := 0;
ELSE
    hbAge := MIN(hbAge + 1, 32000);
END_IF
GVL_Cmd.gwAlive := hbAge < 100;   // 100 * 100 ms = 10 s

// ---------- new command latch ----------
IF (GVL_Cmd.gwCmd.seq <> lastSeq) AND (GVL_Cmd.gwCmd.seq <> 0) THEN
    IF GVL_Cmd.gwPending OR GVL_Cmd.gwAck.busy THEN
        // reject: still executing previous
        GVL_Cmd.gwAck.error := TRUE;
        GVL_Cmd.gwAck.errorId := F_Err(GVL_Cfg.SS_GWCOMMS, GVL_Cfg.ERR_BUSY);
        lastSeq := GVL_Cmd.gwCmd.seq;
        GVL_Cmd.gwAck.seqEcho := lastSeq;
    ELSIF GVL_Cmd.testMode THEN
        GVL_Cmd.gwAck.error := TRUE;
        GVL_Cmd.gwAck.errorId := F_Err(GVL_Cfg.SS_GWCOMMS, GVL_Cfg.ERR_INTERLOCK);
        lastSeq := GVL_Cmd.gwCmd.seq;
        GVL_Cmd.gwAck.seqEcho := lastSeq;
    ELSE
        lastSeq := GVL_Cmd.gwCmd.seq;
        GVL_Cmd.gwAck.seqEcho := lastSeq;
        GVL_Cmd.gwAck.busy := TRUE;
        GVL_Cmd.gwAck.done := FALSE;
        GVL_Cmd.gwAck.error := FALSE;
        GVL_Cmd.gwAck.errorId := 0;
        GVL_Cmd.gwPending := TRUE;
    END_IF
END_IF

// ---------- pack ack ----------
flags := 0;
IF GVL_Cmd.gwAck.busy  THEN flags := flags OR 16#0001; END_IF
IF GVL_Cmd.gwAck.done  THEN flags := flags OR 16#0002; END_IF
IF GVL_Cmd.gwAck.error THEN flags := flags OR 16#0004; END_IF
GVL_Cmd.mbAckRegs[0] := GVL_Cmd.gwAck.seqEcho;
GVL_Cmd.mbAckRegs[1] := flags;
GVL_Cmd.mbAckRegs[2] := DWORD_TO_WORD(GVL_Cmd.gwAck.errorId AND 16#FFFF);
GVL_Cmd.mbAckRegs[3] := DWORD_TO_WORD(SHR(GVL_Cmd.gwAck.errorId, 16));
GVL_Sts.heartbeat := GVL_Sts.heartbeat + 1;
GVL_Cmd.mbAckRegs[4] := GVL_Sts.heartbeat;

// ---------- pack status ----------
GVL_Cmd.mbStsRegs[0] := TO_WORD(TO_UINT(GVL_Sts.mode));
GVL_Cmd.mbStsRegs[1] := BOOL_TO_WORD(GVL_Sts.allHomed)
                      + SHL(BOOL_TO_WORD(GVL_Sts.heatAtSet), 1)
                      + SHL(BOOL_TO_WORD(GVL_Sts.fridgeAtSet), 2)
                      + SHL(BOOL_TO_WORD(GVL_Sts.gwSilent), 3)
                      + SHL(BOOL_TO_WORD(GVL_Cmd.testMode), 4);
FOR z := 0 TO 7 DO
    GVL_Cmd.mbStsRegs[10 + z] := TO_WORD(LREAL_TO_INT(GVL_Sts.aHeat[z].actC * 10.0));
END_FOR
GVL_Cmd.mbStsRegs[18] := TO_WORD(LREAL_TO_INT(GVL_Sts.fridgeActC * 10.0));
FOR gIdx := 0 TO 3 DO
    GVL_Cmd.mbStsRegs[20 + 3 * gIdx]     := TO_WORD(GVL_Sts.aGriddle[gIdx].state);
    GVL_Cmd.mbStsRegs[20 + 3 * gIdx + 1] := TO_WORD(GVL_Sts.aGriddle[gIdx].item);
    GVL_Cmd.mbStsRegs[20 + 3 * gIdx + 2] := TO_WORD(LREAL_TO_INT(GVL_Sts.aGriddle[gIdx].cookElapsedS));
END_FOR
GVL_Cmd.mbStsRegs[32] := TO_WORD(TO_UINT(GVL_Sts.tray.remaining));
GVL_Cmd.mbStsRegs[33] := BOOL_TO_WORD(GVL_Sts.tray.inChamber);
GVL_Cmd.mbStsRegs[34] := TO_WORD(TO_UINT(GVL_Sts.activeAlarms));
GVL_Cmd.mbStsRegs[35] := TO_WORD(TO_UINT(GVL_Sts.carGridStation + 1));
GVL_Cmd.mbStsRegs[36] := UDINT_TO_WORD(GVL_Sts.haccpCount AND 16#FFFF);
// latest HACCP record snapshot (Gateway drains richer log later — TODO ring window)
GVL_Cmd.mbStsRegs[60] := UDINT_TO_WORD(GVL_Sts.lastHaccp.batchId AND 16#FFFF);
GVL_Cmd.mbStsRegs[61] := TO_WORD(GVL_Sts.lastHaccp.item);
GVL_Cmd.mbStsRegs[62] := TO_WORD(TO_UINT(GVL_Sts.lastHaccp.griddleId));
GVL_Cmd.mbStsRegs[63] := TO_WORD(LREAL_TO_INT(GVL_Sts.lastHaccp.platenTopC * 10.0));
GVL_Cmd.mbStsRegs[64] := TO_WORD(LREAL_TO_INT(GVL_Sts.lastHaccp.platenBotC * 10.0));
GVL_Cmd.mbStsRegs[65] := TO_WORD(LREAL_TO_INT(GVL_Sts.lastHaccp.cookS));
GVL_Cmd.mbStsRegs[66] := TO_WORD(GVL_Sts.lastHaccp.result);

